(* IEC 61131-3 sources: ironplc-benchmarks/compat_out (part 63) *)

*)

(* @END_DECLARATION := '0' *)
IF A = 0.0 THEN
	TRIANGLE_A := SQRT((s1+s2+S3) * (s1+s2-S3) * (S2+S3-S1) * (S3+S1-S2)) * 0.25;
ELSE
	TRIANGLE_A := S1 * S2 * SIN(RAD(A)) * 0.5;
END_IF;

(* revision histroy
hm	16. oct 2007	rev 1.0
	original version

hm	22. feb 2008	rev 1.1
	improved performance

hm	10. mar. 2009	rev 1.2
	changed syntax of real constants to 0.0

*)
END_FUNCTION

(* @NESTEDCOMMENTS := 'Yes' *)
(* @PATH := '\/Mathematical\/Vektormathematik' *)
(* @OBJECTFLAGS := '0, 8' *)
(* @SYMFILEFLAGS := '2048' *)
FUNCTION V3_ABS : REAL
VAR_INPUT
	A : Vector_3;
END_VAR

(*
version 1.0	11 dec 2007
programmer 	hugo
tested by		tobias

this function calculates the length of a vectors in a 3 dimensional space

*)
(* @END_DECLARATION := '0' *)
V3_ABS := SQRT(A.X * A.X + A.Y * A.Y + A.Z * A.Z);

(* revision history
hm		11 dec 2007	rev 1.0
	original version

*)
END_FUNCTION

(* @NESTEDCOMMENTS := 'Yes' *)
(* @PATH := '\/Mathematical\/Vektormathematik' *)
(* @OBJECTFLAGS := '0, 8' *)
(* @SYMFILEFLAGS := '2048' *)
FUNCTION V3_ADD : vector_3
VAR_INPUT
	A : Vector_3;
	B : Vector_3;
END_VAR

(*
version 1.0	11 dec 2007
programmer 	hugo
tested by		tobias

this function adds two vectors in a 3 dimensional space

*)
(* @END_DECLARATION := '0' *)
V3_ADD.X := A.X + B.X;
V3_ADD.Y := A.Y + B.Y;
V3_ADD.Z := A.Z + B.Z;

(* revision history
hm		11 dec 2007	rev 1.0
	original version

*)
END_FUNCTION

(* @NESTEDCOMMENTS := 'Yes' *)
(* @PATH := '\/Mathematical\/Vektormathematik' *)
(* @OBJECTFLAGS := '0, 8' *)
(* @SYMFILEFLAGS := '2048' *)
FUNCTION V3_ANG : REAL
VAR_INPUT
	A : Vector_3;
	B : Vector_3;
END_VAR
VAR
	d : REAL;
END_VAR

(*
version 1.1	10. mar. 2009
programmer 	hugo
tested by		tobias

this function calculates the angle between two vectors in a 3 dimensional space

*)
(* @END_DECLARATION := '0' *)
d := V3_ABS(A) * V3_ABS(B);
IF d > 0 THEN
	V3_ANG := ACOS(LIMIT(-1.0, V3_DPRO(A, B) / d,1.0));
END_IF;

(* revision history
hm	11. dec. 2007	rev 1.0
	original version

hm	10. mar. 2009	rev 1.1
	changed syntax of real constants to 0.0

*)
END_FUNCTION

(* @NESTEDCOMMENTS := 'Yes' *)
(* @PATH := '\/Mathematical\/Vektormathematik' *)
(* @OBJECTFLAGS := '0, 8' *)
(* @SYMFILEFLAGS := '2048' *)
FUNCTION V3_DPRO : REAL
VAR_INPUT
	A : Vector_3;
	B : Vector_3;
END_VAR

(*
version 1.0	11 dec 2007
programmer 	hugo
tested by		tobias

this function calculates the dot product of two vectors in 3 dimensional space

*)
(* @END_DECLARATION := '0' *)
V3_DPRO := A.X * B.X + A.Y * B.Y + A.Z * B.Z;

(* revision history
hm		11 dec 2007	rev 1.0
	original version

*)
END_FUNCTION

(* @NESTEDCOMMENTS := 'Yes' *)
(* @PATH := '\/Mathematical\/Vektormathematik' *)
(* @OBJECTFLAGS := '0, 8' *)
(* @SYMFILEFLAGS := '2048' *)
FUNCTION V3_NORM : vector_3
VAR_INPUT
	A : Vector_3;
END_VAR
VAR
	la: REAL;
END_VAR

(*
version 1.1	10. mar. 2009
programmer 	hugo
tested by		tobias

this function generates a vectors with absolute length 1 from a vector A in a 3 dimensional space

*)
(* @END_DECLARATION := '0' *)
la := V3_ABS(A);
IF la > 0.0 THEN
	V3_NORM := V3_SMUL(A, 1.0 / la);
END_IF;

(* revision history
hm	11 dec 2007	rev 1.0
	original version

hm	10. mar. 2009	rev 1.1
	changed syntax of real constants to 0.0

*)
END_FUNCTION

(* @NESTEDCOMMENTS := 'Yes' *)
(* @PATH := '\/Mathematical\/Vektormathematik' *)
(* @OBJECTFLAGS := '0, 8' *)
(* @SYMFILEFLAGS := '2048' *)
FUNCTION V3_NUL : BOOL
VAR_INPUT
	A : Vector_3;
END_VAR

(*
version 1.1	10. mar. 2009
programmer 	hugo
tested by		tobias

this function checks if a vectors in a null Vector

*)
(* @END_DECLARATION := '0' *)
V3_NUL := A.X = 0.0 AND A.Y = 0.0 AND A.Z = 0.0;

(* revision history
hm	12 dec 2007	rev 1.0
	original version

hm	10. mar. 2009	rev 1.1
	changed syntax of real constants to 0.0

*)
END_FUNCTION

(* @NESTEDCOMMENTS := 'Yes' *)
(* @PATH := '\/Mathematical\/Vektormathematik' *)
(* @OBJECTFLAGS := '0, 8' *)
(* @SYMFILEFLAGS := '2048' *)
FUNCTION V3_PAR : BOOL
VAR_INPUT
	A : Vector_3;
	B : Vector_3;
END_VAR

(*
version 1.1	10. mar. 2009
programmer 	hugo
tested by		tobias

this function checks if two vectors in a 3 dimensional space are parallel.
which means the two vectors have the same direction

*)
(* @END_DECLARATION := '0' *)
V3_PAR := V3_ABS(V3_XPRO(A, B)) = 0.0;

(* revision history
hm	11 dec 2007	rev 1.0
	original version

hm	10. mar. 2009	rev 1.1
	changed syntax of real constants to 0.0

*)
END_FUNCTION

(* @NESTEDCOMMENTS := 'Yes' *)
(* @PATH := '\/Mathematical\/Vektormathematik' *)
(* @OBJECTFLAGS := '0, 8' *)
(* @SYMFILEFLAGS := '2048' *)
FUNCTION V3_REV : vector_3
VAR_INPUT
	A : Vector_3;
END_VAR

(*
version 1.0	11 dec 2007
programmer 	hugo
tested by		tobias

this function reverses a vector in a 3 dimensional space

*)
(* @END_DECLARATION := '0' *)
V3_REV.X := -A.X;
V3_REV.Y := -A.Y;
V3_REV.Z := -A.Z;

(* revision history
hm		11 dec 2007	rev 1.0
	original version

*)
END_FUNCTION

(* @NESTEDCOMMENTS := 'Yes' *)
(* @PATH := '\/Mathematical\/Vektormathematik' *)
(* @OBJECTFLAGS := '0, 8' *)
(* @SYMFILEFLAGS := '2048' *)
FUNCTION V3_SMUL : vector_3
VAR_INPUT
	A : Vector_3;
	M : REAL;
END_VAR

(*
version 1.0	11 dec 2007
programmer 	hugo
tested by		tobias

this function multiplies a vectors in a 3 dimensional space with a skalar M

*)
(* @END_DECLARATION := '0' *)
V3_SMUL.X := A.X * M;
V3_SMUL.Y := A.Y * M;
V3_SMUL.Z := A.Z * M;

(* revision history
hm		11 dec 2007	rev 1.0
	original version

*)
END_FUNCTION

(* @NESTEDCOMMENTS := 'Yes' *)
(* @PATH := '\/Mathematical\/Vektormathematik' *)
(* @OBJECTFLAGS := '0, 8' *)
(* @SYMFILEFLAGS := '2048' *)
FUNCTION V3_SUB : vector_3
VAR_INPUT
	A : Vector_3;
	B : Vector_3;
END_VAR

(*
version 1.0	11 dec 2007
programmer 	hugo
tested by		tobias

this function subtracts two vectors in a 3 dimensional space
V3_SUB = A - B

*)
(* @END_DECLARATION := '0' *)
V3_SUB.X := A.X - B.X;
V3_SUB.Y := A.Y - B.Y;
V3_SUB.Z := A.Z - B.Z;

(* revision history
hm		11 dec 2007	rev 1.0
	original version

*)
END_FUNCTION

(* @NESTEDCOMMENTS := 'Yes' *)
(* @PATH := '\/Mathematical\/Vektormathematik' *)
(* @OBJECTFLAGS := '0, 8' *)
(* @SYMFILEFLAGS := '2048' *)
FUNCTION V3_XANG : REAL
VAR_INPUT
	A : Vector_3;
END_VAR
VAR
	la: REAL;
END_VAR

(*
version 1.1	10. mar. 2009
programmer 	hugo
tested by		tobias

this function calculates the angle between the X-axis and a vectors in a 3 dimensional space

*)
(* @END_DECLARATION := '0' *)
la := V3_ABS(a);
IF la > 0.0 THEN
	V3_XANG := ACOS(A.X / la);
END_IF;

(* revision history
hm	11 dec 2007	rev 1.0
	original version

hm	10. mar. 2009	rev 1.1
	changed syntax of real constants to 0.0

*)
END_FUNCTION

(* @NESTEDCOMMENTS := 'Yes' *)
(* @PATH := '\/Mathematical\/Vektormathematik' *)
(* @OBJECTFLAGS := '0, 8' *)
(* @SYMFILEFLAGS := '2048' *)
FUNCTION V3_XPRO : vector_3
VAR_INPUT
	A : Vector_3;
	B : Vector_3;
END_VAR

(*
version 1.0	11 dec 2007
programmer 	hugo
tested by		tobias

this function adds two vectors in a 3 dimensional space

*)
(* @END_DECLARATION := '0' *)
V3_XPRO.X := A.Y * B.Z - A.Z * B.Y;
V3_XPRO.Y := A.Z * B.X - A.X * B.Z;
V3_XPRO.Z := A.X * B.Y - A.Y * B.X;

(* revision history
hm		11 dec 2007	rev 1.0
	original version

*)
END_FUNCTION

(* @NESTEDCOMMENTS := 'Yes' *)
(* @PATH := '\/Mathematical\/Vektormathematik' *)
(* @OBJECTFLAGS := '0, 8' *)
(* @SYMFILEFLAGS := '2048' *)
FUNCTION V3_YANG : REAL
VAR_INPUT
	A : Vector_3;
END_VAR
VAR
	la: REAL;
END_VAR

(*
version 1.1	10. mar. 2009
programmer 	hugo
tested by		tobias

this function calculates the angle between the Y-axis and a vectors in a 3 dimensional space

*)
(* @END_DECLARATION := '0' *)
la := V3_ABS(a);
IF la > 0.0 THEN
	V3_YANG := ACOS(A.Y / la);
END_IF;

(* revision history
hm	11 dec 2007	rev 1.0
	original version

hm	10. mar. 2009	rev 1.1
	changed syntax of real constants to 0.0

*)
END_FUNCTION

(* @NESTEDCOMMENTS := 'Yes' *)
(* @PATH := '\/Mathematical\/Vektormathematik' *)
(* @OBJECTFLAGS := '0, 8' *)
(* @SYMFILEFLAGS := '2048' *)
FUNCTION V3_ZANG : REAL
VAR_INPUT
	A : Vector_3;
END_VAR
VAR
	la: REAL;
END_VAR

(*
version 1.1	10. mar. 2009
programmer 	hugo
tested by		tobias

this function calculates the angle between the Z-axis and a vectors in a 3 dimensional space

*)
(* @END_DECLARATION := '0' *)
la := V3_ABS(a);
IF la > 0.0 THEN
	V3_ZANG := ACOS(A.Z / la);
END_IF;

(* revision history
hm	11 dec 2007	rev 1.0
	original version

hm	10. mar. 2009	rev 1.1
	changed syntax of real constants to 0.0

*)
END_FUNCTION

(* @NESTEDCOMMENTS := 'Yes' *)
(* @PATH := '\/Mathematical' *)
(* @OBJECTFLAGS := '0, 8' *)
(* @SYMFILEFLAGS := '2048' *)
FUNCTION ACOSH : REAL
VAR_INPUT
	X : REAL;
END_VAR

(*
version 1.3	10. mar. 2009
programmer 	hugo
tested by		tobias

this function calculates the arcus cos hyperbolicus

*)
(* @END_DECLARATION := '0' *)
ACOSH := LN(SQRT(X * X - 1.0) + X);

(* revision history
hm		12 jan 2007	rev 1.0
	original version

hm		2. dec 2007	rev 1.1
	changed code for better performance

hm	16. mar. 2007		rev 1.2
	changed sequence of calculations to improve performance

hm	10. mar. 2009		rev 1.3
	real constants updated to new systax using dot

*)
END_FUNCTION

(* @NESTEDCOMMENTS := 'Yes' *)
(* @PATH := '\/Mathematical' *)
(* @OBJECTFLAGS := '0, 8' *)
(* @SYMFILEFLAGS := '2048' *)
FUNCTION ACOTH : REAL
VAR_INPUT
	X : REAL;
END_VAR

(*
version 1.2	10. mar. 2009
programmer 	hugo
tested by		tobias

this function calculates the arcus cotangens hyperbolicus

*)
(* @END_DECLARATION := '0' *)
ACOTH := LN((x+1.0)/(x-1.0))*0.5;

(* revision history
hm		12 jan 2007	rev 1.0
	original version

hm		5. jan 2008	rev 1.1
	improved code for better performance

hm	10. mar. 2009		rev 1.2
	real constants updated to new systax using dot

*)
END_FUNCTION

(* @NESTEDCOMMENTS := 'Yes' *)
(* @PATH := '\/Mathematical' *)
(* @OBJECTFLAGS := '0, 8' *)
(* @SYMFILEFLAGS := '2048' *)
FUNCTION AGDF : REAL
VAR_INPUT
	X : REAL;
END_VAR

(*
version 1.1	10. mar. 2009
programmer 	hugo
tested by		tobias

this function calculates the inverse Gudermannian function.

*)
(* @END_DECLARATION := '0' *)
AGDF := LN((1.0 + SIN(X)) / COS(X));

(* comment
the current implementation gives sufficient accuracy only up to X = 1.57 or an output > 10.
is X closer to PI/2 then the function is more and more unreliable
*)

(* revision history
hm	27. apr. 2008	rev 1.0
	original version

hm	10. mar. 2009	rev 1.1
	real constants updated to new systax using dot

*)

END_FUNCTION

(* @NESTEDCOMMENTS := 'Yes' *)
(* @PATH := '\/Mathematical' *)
(* @OBJECTFLAGS := '0, 8' *)
(* @SYMFILEFLAGS := '2048' *)
FUNCTION ASINH : REAL
VAR_INPUT
	X : REAL;
END_VAR

(*
version 1.3	10. mar 2009
programmer 	hugo
tested by		tobias

this function calculates the arcus sin hyperbolicus

*)
(* @END_DECLARATION := '0' *)
ASINH := LN(SQRT(X * X + 1.0)+X);

(* revision history
hm		12 jan 2007	rev 1.0
	original version

hm		2. dec 2007	rev 1.1
	changed code for better performance

hm		16.3. 2007		rev 1.2
	changed sequence of calculations to improve performance

hm	10. mar. 2009		rev 1.3
	real constants updated to new systax using dot

*)
END_FUNCTION

(* @NESTEDCOMMENTS := 'Yes' *)
(* @PATH := '\/Mathematical' *)
(* @OBJECTFLAGS := '0, 8' *)
(* @SYMFILEFLAGS := '2048' *)
FUNCTION ATANH : REAL
VAR_INPUT
	X : REAL;
END_VAR

(*
version 1.2	10. mar. 2009
programmer 	hugo
tested by		tobias

this function calculates the arcus tangens hyperbolicus

*)
(* @END_DECLARATION := '0' *)
ATANH := LN((1.0 + x)/(1.0 - x)) * 0.5;

(* revision history
hm		12 jan 2007	rev 1.0
	original version

hm		5. jan 2008	rev 1.1
	improved code for better performance

hm	10. mar. 2009		rev 1.2
	real constants updated to new systax using dot

*)

END_FUNCTION

(* @NESTEDCOMMENTS := 'Yes' *)
(* @PATH := '\/Mathematical' *)
(* @OBJECTFLAGS := '0, 8' *)
(* @SYMFILEFLAGS := '2048' *)
FUNCTION BETA : REAL
VAR_INPUT
	X : REAL;
	Y : REAL;
END_VAR

(*
version 1.0	26. oct. 2008
programmer 	hugo
tested by		oscat

this function calculates the beta function for real number > 0.

*)
(* @END_DECLARATION := '0' *)
BETA := GAMMA(X) * GAMMA(Y) / GAMMA(x + y);

(* revision history
hm	26. oct. 2008	rev 1.0
	original version

*)
END_FUNCTION

(* @NESTEDCOMMENTS := 'Yes' *)
(* @PATH := '\/Mathematical' *)
(* @OBJECTFLAGS := '0, 8' *)
(* @SYMFILEFLAGS := '2048' *)
FUNCTION BINOM : DINT
VAR_INPUT
	N : INT;
	K : INT;
END_VAR

VAR
	i: INT;
END_VAR

(*
version 1.0	25. oct. 2008
programmer 	hugo
tested by		tobias

this function calculates the binomialkoefficient (N over k)

*)
(* @END_DECLARATION := '0' *)
IF 2 * K > n THEN
	k := n - k;
END_IF;
IF k > n THEN
	RETURN;
ELSIF k = 0 OR k = n THEN
	BINOM := 1;
ELSIF k = 1 THEN
	BINOM := n;
ELSE
	BINOM := n;
	n := n + 1;
	FOR i := 2 TO k DO
		BINOM := BINOM * (n - i) / i;
	END_FOR;
END_IF;

(*
binomialkoeffizient(n, k)
1  wenn k = 0 return 1
2  wenn 2k > n
3      dann f�hre aus ergebnis \leftarrow binomialkoeffizient(n, n-k)
4  sonst f�hre aus ergebnis \leftarrow n
5          von i \leftarrow 2 bis k
6              f�hre aus ergebnis \leftarrow ergebnis \cdot (n + 1 - i)
7                        ergebnis \leftarrow ergebnis : i
8  return ergebnis
*)

(* revision history
hm	25. oct. 2008	rev 1.0
	original version

*)
END_FUNCTION

(* @NESTEDCOMMENTS := 'Yes' *)
(* @PATH := '\/Mathematical' *)
(* @OBJECTFLAGS := '0, 8' *)
(* @SYMFILEFLAGS := '2048' *)
FUNCTION CAUCHY : REAL
VAR_INPUT
	X : REAL;
	T : REAL;
	U : REAL;
END_VAR
VAR
	tmp: REAL;
END_VAR

(*
version 1.0	26. oct. 2008
programmer 	hugo
tested by		tobias

this function calculates the Cauchy distribution function

*)
(* @END_DECLARATION := '0' *)
tmp := x - t;
CAUCHY := math.PI_INV * U / (U*U + tmp*tmp);

(* revision hisdtory
hm	26. oct. 2008	rev 1.0
	original version

*)
END_FUNCTION

(* @NESTEDCOMMENTS := 'Yes' *)
(* @PATH := '\/Mathematical' *)
(* @OBJECTFLAGS := '0, 8' *)
(* @SYMFILEFLAGS := '2048' *)
FUNCTION CAUCHYCD : REAL
VAR_INPUT
	X : REAL;
	T : REAL;
	U : REAL;
END_VAR

(*
version 1.0	26. oct. 2008
programmer 	hugo
tested by		tobias

this function calculates the Cauchy distribution function

*)
(* @END_DECLARATION := '0' *)
CAUCHYCD := 0.5 + math.PI_INV * ATAN((X - T) / U);

(* revision hisdtory
hm	26. oct. 2008	rev 1.0
	original version

*)
END_FUNCTION

(* @NESTEDCOMMENTS := 'Yes' *)
(* @PATH := '\/Mathematical' *)
(* @OBJECTFLAGS := '0, 8' *)
(* @SYMFILEFLAGS := '2048' *)
FUNCTION CEIL : INT
VAR_INPUT
	X : REAL;
END_VAR

(*
version 1.1	21. mar. 2008
programmer 	hugo
tested by	tobias

This is a rounding function which returns the smallest possible integer which is greater or equal to X.
ceil(3.14) = 4
ceil(-3.14) = -3

*)

(* @END_DECLARATION := '0' *)
CEIL := REAL_TO_INT(x);
IF CEIL < X THEN
	CEIL := CEIL + 1;
END_IF;

(* revision history
hm	7. feb. 2007	rev 1.0
	original version

hm	21. mar. 2008	rev 1.1
	use REAL_TO_INT instead of trunc for compatibility reasons

*)

END_FUNCTION

(* @NESTEDCOMMENTS := 'Yes' *)
(* @PATH := '\/Mathematical' *)
(* @OBJECTFLAGS := '0, 8' *)
(* @SYMFILEFLAGS := '2048' *)
FUNCTION CEIL2 : DINT
VAR_INPUT
	X : REAL;
END_VAR

(*
version 1.3	10. mar. 2009
programmer 	hugo
tested by		tobias

This is a rounding function which returns the smallest possible integer which is greater or equal to X.
ceil2(3.14) = 4
ceil2(-3.14) = -3

*)

(* @END_DECLARATION := '0' *)
CEIL2 := REAL_TO_DINT(X);
IF DINT_TO_REAL(CEIL2) < X THEN
	CEIL2 := CEIL2 + 1;
END_IF;

(* revision history
hm	21. mar. 2008	rev 1.0
	original version

hm	4. apr. 2008	rev 1.1
	added type conversion to avoid warnings under codesys 3.0

hm	30. jun. 2008	rev 1.2
	added type conversion to avoid warnings under codesys 3.0

hm	10. mar. 2009	rev 1.3
	use correct statement real_to_DINT

*)

END_FUNCTION

(* @NESTEDCOMMENTS := 'Yes' *)
(* @PATH := '\/Mathematical' *)
(* @OBJECTFLAGS := '0, 8' *)
(* @SYMFILEFLAGS := '2048' *)
FUNCTION CMP : BOOL
VAR_INPUT
	X,Y : REAL;
	N : INT;
END_VAR
VAR
	tmp : REAL;
END_VAR

(*
	version 1.1	10. mar. 2009
	programmer 	hugo
	tested by		tobias

this function checks two inputs x and y if they are identical with the first N digits
example : cmp(3.141516,3.141517,6 is true.

*)
(* @END_DECLARATION := '0' *)
tmp := ABS(x);
IF tmp > 0.0 THEN
	tmp := EXP10(INT_TO_REAL(FLOOR(LOG(tmp))-N+1));
ELSE
	tmp := EXP10(tmp);
END_IF;
CMP := ABS(X - Y) < tmp;

(* revision history
hm	12. mar. 2008	rev 1.0
	original version

hm	10. mar. 2009	rev 1.1
	added type conversion for compatibility reasons
*)

END_FUNCTION

(* @NESTEDCOMMENTS := 'Yes' *)
(* @PATH := '\/Mathematical' *)
(* @OBJECTFLAGS := '0, 8' *)
(* @SYMFILEFLAGS := '2048' *)
FUNCTION COSH : REAL
VAR_INPUT
	X : REAL;
END_VAR
VAR
	t: REAL;
END_VAR

(*
version 1.3	10. mar. 2009
programmer 	hugo
tested by		tobias

this function calculates the cos hyperbolicus

*)
(* @END_DECLARATION := '0' *)
T := EXP(X);
COSH := (1.0 / T + T) * 0.5;

(* revision histroy
hm	12.1.2007	rev 1.0
	original version

hm	1.12.2007	rev 1.1
	changed code to improve performance

hm	5. jan 2008	rev 1.2
	further performance improvement

hm	10. mar. 2009	rev 1.3
	real constants updated to new systax using dot
*)
END_FUNCTION

(* @NESTEDCOMMENTS := 'Yes' *)
(* @PATH := '\/Mathematical' *)
(* @OBJECTFLAGS := '0, 8' *)
(* @SYMFILEFLAGS := '2048' *)
FUNCTION COTH : REAL
VAR_INPUT
	X : REAL;
END_VAR

(*
version 1.4	10. mar. 2009
programmer 	hugo
tested by		tobias

this function calculates the cotangens hyperbolicus

*)
(* @END_DECLARATION := '0' *)
IF X > 20.0 THEN
	COTH :=1.0;
ELSIF X < -20.0 THEN
	COTH := -1.0;
ELSE
	COTH := 1.0 + 2.0 / (EXP(X * 2.0) - 1.0);
END_IF;

(* revision histroy
hm		12.1.2007	rev 1.0
	original version

hm	1.12.2007		rev 1.1
	changed code to improve performance

hm	8. jan 2008	rev 1.2
	further improvement in performance

hm	10. mar 2008	rev 1.3
	extended range of valid inputs to +/- INV
	changed formula for better accuracy

hm	10. mar. 2009	rev 1.4
	real constants updated to new systax using dot
*)
END_FUNCTION

(* @NESTEDCOMMENTS := 'Yes' *)
(* @PATH := '\/Mathematical' *)
(* @OBJECTFLAGS := '0, 8' *)
(* @SYMFILEFLAGS := '2048' *)
FUNCTION D_TRUNC : DINT
VAR_INPUT
	X : REAL;
END_VAR

(*
version 1.2	10. mar. 2009
programmer 	hugo
tested by		oscat

d_trunc truncates a real to a dint 1.5 will be 1 and -1.5 will be -1
d_trunc is necessary because many systems do not offer a trunc to a dint
also real_to_dint will not deliver the same result on different systems

*)

(* @END_DECLARATION := '0' *)
D_TRUNC := REAL_TO_DINT(X);
IF X > 0.0 THEN
	IF DINT_TO_REAL(D_TRUNC) > X THEN D_TRUNC := D_TRUNC - 1; END_IF;
ELSE
	IF DINT_TO_REAL(D_TRUNC) < X THEN D_TRUNC := D_TRUNC + 1; END_IF;
END_IF;

(* for systems that support a dint truncation this routine can be replaced by trunc() *)

(* revision history
hm	21. mar. 2008	rev 1.0
	original version

hm	31. oct. 2008	rev 1.1
	optimized performance

hm	10. mar. 2009	rev 1.2
	real constants updated to new systax using dot
*)
END_FUNCTION

(* @NESTEDCOMMENTS := 'Yes' *)
(* @PATH := '\/Mathematical' *)
(* @OBJECTFLAGS := '0, 8' *)
(* @SYMFILEFLAGS := '2048' *)
FUNCTION DEC1 : INT
VAR_INPUT
	X : INT;
	N : INT;
END_VAR

(*
version 1.1	27. oct. 2008
programmer 	hugo
tested by	oscat

This is a decrement function which decrements the variable X by 1 and if 0 is reached, it begins with N-1 again.
_dec1(X,3) will generate 2,1,0,2,...

*)
(* @END_DECLARATION := '0' *)
IF X = 0 THEN
	DEC1 := N - 1;
ELSE
	DEC1 := X - 1;
END_IF;

(* this is a very elegant version but 50% slower
X := (X - 1 + N) MOD N;
*)

(* revision history
hm	13. oct. 2008	rev 1.0
	original version

hm	27. oct. 2008	rev 1.1
	added statement to return value for compatibility reasons

*)
END_FUNCTION

(* @NESTEDCOMMENTS := 'Yes' *)
(* @PATH := '\/Mathematical' *)
(* @OBJECTFLAGS := '0, 8' *)
(* @SYMFILEFLAGS := '2048' *)
FUNCTION DEG : REAL
VAR_INPUT
	rad : REAL;
END_VAR

(*
version 1.2	10. mar. 2009
programmer 	hugo
tested by		tobias

this function converts degrees into Radiant
execution time on wago 750 - 841 =  10  us
*)
(* @END_DECLARATION := '0' *)
DEG := MODR(57.29577951308232 * RAD, 360.0);

(* revision history
hm	4. aug 2006	rev 1.0
	original version

hm 16. oct 2007	rev 1.1
	added modr statement which prohibits deg to become bigger than 360

hm	10. mar. 2009	rev 1.2
	real constants updated to new systax using dot
*)
END_FUNCTION

(* @NESTEDCOMMENTS := 'Yes' *)
(* @PATH := '\/Mathematical' *)
(* @OBJECTFLAGS := '0, 8' *)
(* @SYMFILEFLAGS := '2048' *)
FUNCTION DIFFER : BOOL
VAR_INPUT
	in1 : REAL;
	in2 : REAL;
	X : REAL;
END_VAR

(*
version 1.1	16 mar 2008
programmer 	hugo
tested by		tobias

this function checks if in1 differs more then x from in2
the output is true if abs(in1-in2) > X

*)
(* @END_DECLARATION := '0' *)
DIFFER := ABS(in1 - in2) > X;

(* revision history
hm		8. oct 2006		rev 1.0
	original version

hm		16. mar 2008	rev 1.1
	improverd code for performance

*)
END_FUNCTION

(* @NESTEDCOMMENTS := 'Yes' *)
(* @PATH := '\/Mathematical' *)
(* @OBJECTFLAGS := '0, 8' *)
(* @SYMFILEFLAGS := '2048' *)
FUNCTION ERF : REAL
VAR_INPUT
	X : REAL;
END_VAR
VAR
	x2 : REAL;
	ax2 : REAL;
END_VAR

(*
version 1.3	10. mar. 2009
programmer 	hugo
tested by		tobias

this function calculates the erf (error) function.

*)
(* @END_DECLARATION := '0' *)
x2 := X*X;
ax2 := 0.147 * x2 + 1.0;
ERF := SQRT(1.0 - EXP(-X2 * ((0.27323954473516 + aX2)/(ax2)))) * SGN(x);

(* revision history
hm	7. apr. 2008	rev 1.0
	original version

hm	30. jun. 2008	rev 1.1
	added type conversions to avoid warnings under codesys 3.0

hm	25. oct. 2008	rev 1.2
	new code using new algorithm

hm	10. mar. 2009	rev 1.3
	real constants updated to new systax using dot
*)
END_FUNCTION

(* @NESTEDCOMMENTS := 'Yes' *)
(* @PATH := '\/Mathematical' *)
(* @OBJECTFLAGS := '0, 8' *)
(* @SYMFILEFLAGS := '2048' *)
FUNCTION ERFC : REAL
VAR_INPUT
	X : REAL;
END_VAR

(*
version 1.1	10. mar. 2009
programmer 	hugo
tested by		tobias

this function calculates the inverse erf (error) function.

*)
(* @END_DECLARATION := '0' *)
ERFC := 1.0 - ERF(X);

(* revision history
hm	7. apr. 2008	rev 1.0
	original version

hm	10. mar. 2009	rev 1.1
	real constants updated to new systax using dot

*)
END_FUNCTION

(* @NESTEDCOMMENTS := 'Yes' *)
(* @PATH := '\/Mathematical' *)
(* @OBJECTFLAGS := '0, 8' *)
(* @SYMFILEFLAGS := '2048' *)
FUNCTION EVEN : BOOL
VAR_INPUT
	in : DINT;
END_VAR

(*
version 1.1	1 dec 2007
programmer 	hugo
tested by		tobias

this function chacks an input for even  value
the output is true if the input is even.
execution time on wago 750 - 841 =  10  us
*)
(* @END_DECLARATION := '0' *)
EVEN := NOT in.0;

(* revision history
hm	1. oct 2006	rev 1.0
	ORIGINAL VERSION

hm	01.12.2007	rev 1.1
	changed code for improved performance

hm	21. mar. 2008	rev 1.2
	changed type of input IN from INT to DINT
*)
END_FUNCTION

(* @NESTEDCOMMENTS := 'Yes' *)
(* @PATH := '\/Mathematical' *)
(* @OBJECTFLAGS := '0, 8' *)
(* @SYMFILEFLAGS := '2048' *)
FUNCTION EXP10 : REAL
VAR_INPUT
	X : REAL;
END_VAR

(*
version 1.0	 2 dec 2007
programmer 	hugo
tested by		tobias

this function calculates the exponent to the basis 10
exp10(3) = 1000

*)
(* @END_DECLARATION := '0' *)
EXP10 := EXP(X * 2.30258509299405);

(* revision history
hm	2. dec 2007		rev 1.0
	original version

*)
END_FUNCTION

(* @NESTEDCOMMENTS := 'Yes' *)
(* @PATH := '\/Mathematical' *)
(* @OBJECTFLAGS := '0, 8' *)
(* @SYMFILEFLAGS := '2048' *)
FUNCTION EXPN : REAL
VAR_INPUT
	X : REAL;
	N : INT;
END_VAR
VAR
	sign: BOOL;
END_VAR

(*
version 1.2	10. mar. 2009
programmer 	hugo
tested by		oscat

this function calculates X to the power of N (Y = X^N) whilke N is an integer
especially on CPU's without a floating point unit this algorythm is about 30 times faster then the IEC standard EXPT() Function

*)
(* @END_DECLARATION := '0' *)
sign := n.15;
N := ABS(N);
IF N.0 THEN EXPN := X; ELSE EXPN := 1.0; END_IF;
N := SHR(N,1);
WHILE N > 0 DO
   X := X * X;
   IF N.0 THEN EXPN := EXPN * X; END_IF;
   N := SHR(N,1);
END_WHILE;
IF sign THEN EXPN := 1.0 / EXPN; END_IF;

(* revision history
hm	4. dec 2007	rev 1.0
	original version

hm	22. oct. 2008	rev 1.1
	optimized code

hm	10. mar. 2009	rev 1.2
	removed nested comments
	real constants updated to new systax using dot

*)
END_FUNCTION

(* @NESTEDCOMMENTS := 'Yes' *)
(* @PATH := '\/Mathematical' *)
(* @OBJECTFLAGS := '0, 8' *)
(* @SYMFILEFLAGS := '2048' *)
FUNCTION FACT : DINT
VAR_INPUT
	X : INT;
END_VAR

(*
version 1.5	26. mar. 2011
programmer 	hugo
tested by		tobias

this function calculates the factorial of x

if the input is negative or higher then 12 the output will be -1.

*)
(* @END_DECLARATION := '0' *)
IF X >= 0 AND X <= 12 THEN
	FACT := math.FACTS[X];
ELSE
	FACT := -1;
END_IF;

(* working code without array
IF X > 12 OR X < 0 THEN
	FACT := -1;
ELSIF X < 7 THEN
	FACT := 1;
	FOR i := 2 TO X DO
		FACT := FACT * i;
	END_FOR;
ELSE
	FACT := 5040;
	FOR i := 8 TO X DO
		FACT := FACT * i;
	END_FOR;
END_IF;
*)

(* revision history
hm 4.3.2007		rev 1.1
	changed a critical error where while loop was indefinite.

hm	10.12.2007	rev 1.2
	start value for i has changed to 2 for better performance

hm	10. mar 2008	rev 1.3
	changed output of fact to dint to allow bigger values

hm	27. oct. 2008	rev 1.4
	optimized code

hm	26. mar. 2011	rev 1.5
	using array math.facts
*)
END_FUNCTION

(* @NESTEDCOMMENTS := 'Yes' *)
(* @PATH := '\/Mathematical' *)
(* @OBJECTFLAGS := '0, 8' *)
(* @SYMFILEFLAGS := '2048' *)
FUNCTION FIB : DINT
VAR_INPUT
	X : INT;
END_VAR
VAR
	t1, t2: DINT;
END_VAR

(*
version 1.3	26. mar. 2008
programmer 	hugo
tested by		tobias

this function calculates the fibonacci sequence

*)
(* @END_DECLARATION := '0' *)
IF X < 0 OR X > 46 THEN
	FIB := -1;
ELSIF x < 2 THEN
	FIB := X;
	RETURN;
ELSE
	(* the fibonacci number is the sum of the two suceeding fibonaci numbers *)
	(* we store the numbers alternatively in t1 and t2 depending on pt *)
	t2 := 1;
	WHILE X > 3 DO
		X := X-2;
		t1 := t1 + t2;
		t2 := t1 + t2;
	END_WHILE;
	IF X > 2 THEN t1 := t1 + t2; END_IF;
	fib := t1 + t2;
END_IF;

(* alternative code for very big numbers

IF X < 31 THEN
	fib := 0.4472136 * (expn(1.618034,X) - expn(-0.618034,X));
ELSE
	fib := 0.4472133 * expn(1.618034,X);
END_IF;

*)

(* revision history
hm		27. dec 2007	rev 1.0
	original version

hm		2. jan 2008	rev 1.1
	deleted unused variable pt

hm		10. mar 2008	rev 1.2
	changed output to dint instead of real

hm		26. mar. 2008	rev 1.3
	function now returns -1 for input < 0 or > 46

*)
END_FUNCTION

(* @NESTEDCOMMENTS := 'Yes' *)
(* @PATH := '\/Mathematical' *)
(* @OBJECTFLAGS := '0, 8' *)
(* @SYMFILEFLAGS := '2048' *)
FUNCTION FLOOR : INT
VAR_INPUT
	X : REAL;
END_VAR

(*
version 1.1	21. mar. 2008
programmer 	hugo
tested by		tobias

This is a rounding function which returns the biggest possible integer which is less or equal to X.
floor(3.14) = 3
floor(-3.14) = -4

*)

(* @END_DECLARATION := '0' *)
FLOOR := REAL_TO_INT(X);
IF FLOOR > X THEN
	FLOOR := FLOOR - 1;
END_IF;

(* revision history
hm		7. feb 2007		rev 1.0
	originlal version

hm		21. mar. 2008	rev 1.1
	replaced trunc with real_to_int for compatibility reasons

*)
END_FUNCTION

(* @NESTEDCOMMENTS := 'Yes' *)
(* @PATH := '\/Mathematical' *)
(* @OBJECTFLAGS := '0, 8' *)
(* @SYMFILEFLAGS := '2048' *)
FUNCTION FLOOR2 : DINT
VAR_INPUT
	X : REAL;
END_VAR

(*
version 1.1	4. apr. 2008
programmer 	hugo
tested by		tobias

This is a rounding function which returns the biggest possible integer which is less or equal to X.
floor2(3.14) = 3
floor2(-3.14) = -4

*)

(* @END_DECLARATION := '0' *)
FLOOR2 := REAL_TO_DINT(X);
IF DINT_TO_REAL(FLOOR2) > X THEN
	FLOOR2 := FLOOR2 - 1;
END_IF;

(* revision history
hm	21. mar. 2008	rev 1.0
	originlal version

hm	4. apr. 2008	rev 1.1
	added type conversion to avoid warnings under codesys 3.0
*)
END_FUNCTION

(* @NESTEDCOMMENTS := 'Yes' *)
(* @PATH := '\/Mathematical' *)
(* @OBJECTFLAGS := '0, 8' *)
(* @SYMFILEFLAGS := '2048' *)
FUNCTION FRACT : REAL
VAR_INPUT
	x : REAL;
END_VAR

(*
version 1.3	10. mar. 2009
programmer 	hugo
tested by		tobias

this function returns the fraction of a real number
fract(3.14) = 0.14

*)
(* @END_DECLARATION := '0' *)
IF ABS(x) < 2.0E9 THEN
	FRACT := x - DINT_TO_REAL(D_TRUNC(x));
ELSE
	FRACT := 0.0;
END_IF;

(* revision history
hm	4. aug 2006	rev 1.0
	original version

hm	11. mar 2008	rev 1.1
	added dint_to_real for compatibility reasons
	now returns 0 for number > 2e9
	changed input to x

hm	21. mar. 2008	rev 1.2
	use D_trunc instead of TRUNC for compatibility reasons

hm	10. mar. 2009	rev 1.3
	real constants updated to new systax using dot

*)
END_FUNCTION

(* @NESTEDCOMMENTS := 'Yes' *)
(* @PATH := '\/Mathematical' *)
(* @OBJECTFLAGS := '0, 8' *)
(* @SYMFILEFLAGS := '2048' *)
FUNCTION GAMMA : REAL
VAR_INPUT
	X : REAL;
END_VAR

(*
version 1.3	10. mar. 2009
programmer 	hugo
tested by		oscat

this function calculates the stirling function which is an approximation for the gamma function

*)
(* @END_DECLARATION := '0' *)
IF x > 0.0 THEN
	GAMMA := SQRT(math.PI2 / X) * EXPT(math.E_INV * (x + 1.0 / (12.0 * x - 0.1 / X)), X);
END_IF;

(* the stirling formula is not very accurate for small values of X
IF X >=0 THEN GAMMA := SQRT(math.PI2 * X) * EXPT(X / math.E, X); END_IF;
*)

(* revision history
hm	10.12.2007	rev 1.0
	original version

hm	18. oct. 2008	rev 1.1
	using math constants

hm	26. oct. 2008	rev 1.2
	using new formula with better accuracy

hm	10. mar. 2009	rev 1.3
	real constants updated to new systax using dot

*)
END_FUNCTION

(* @NESTEDCOMMENTS := 'Yes' *)
(* @PATH := '\/Mathematical' *)
(* @OBJECTFLAGS := '0, 8' *)
(* @SYMFILEFLAGS := '2048' *)
FUNCTION GAUSS : REAL
VAR_INPUT
	X : REAL;
	U : REAL;
	SI: REAL;
END_VAR
VAR
	temp: REAL;
	si_inv: REAL;
END_VAR

(*
version 1.2	10. mar. 2009
programmer 	hugo
tested by		tobias

this function calculates the gaussian density function

*)
(* @END_DECLARATION := '0' *)
temp := X - U;
si_inv := 1.0  / si;
GAUSS := EXP(Temp * Temp * si_inv * si_inv * - 0.5) * 0.39894228 * si_inv;

(* revision hisdtory
hm	6. apr. 2008	rev 1.0
	original version

hm	27. oct. 2008	rev 1.1
	optimized performance

hm	10. mar. 2009	rev 1.2
	real constants updated to new systax using dot

*)
END_FUNCTION

(* @NESTEDCOMMENTS := 'Yes' *)
(* @PATH := '\/Mathematical' *)
(* @OBJECTFLAGS := '0, 8' *)
(* @SYMFILEFLAGS := '2048' *)
FUNCTION GAUSSCD : REAL
VAR_INPUT
	X : REAL;
	U : REAL;
	SI: REAL;
END_VAR

(*
version 1.1	10. mar. 2009
programmer 	hugo
tested by		tobias

this function calculates the gaussian cumulative distribution function

*)
(* @END_DECLARATION := '0' *)
GAUSSCD := (ERF((X - U) / (SI * 1.414213562)) + 1.0) * 0.5;

(* revision hisdtory
hm	6. apr. 2008	rev 1.0
	original version

hm	10. mar. 2009	rev 1.1
	real constants updated to new systax using dot

*)
END_FUNCTION

(* @NESTEDCOMMENTS := 'Yes' *)
(* @PATH := '\/Mathematical' *)
(* @OBJECTFLAGS := '0, 8' *)
(* @SYMFILEFLAGS := '2048' *)
FUNCTION GCD : INT
VAR_INPUT
	A : DINT;
	B : DINT;
END_VAR
VAR
	t: DINT;
END_VAR

(*
version 1.0	19. jan. 2011
programmer 	hugo
tested by	tobias

this function calculates the gretaest common divisor of two numbers A and B

*)
(* @END_DECLARATION := '0' *)
IF A = 0 THEN
	GCD := DINT_TO_INT(ABS(B));
ELSIF B = 0 THEN
	GCD := DINT_TO_INT(ABS(A));
ELSE
	A := ABS(A);
	B := ABS(B);
	GCD := 1;
	WHILE NOT(A.0 OR B.0) DO
		A := SHR(A,1);
		B := SHR(B,1);
		GCD := SHL(GCD,1);
	END_WHILE;
	WHILE A > 0 DO
		IF NOT(A.0) THEN A := SHR(A,1);
		ELSIF NOT(B.0) THEN B := SHR(B,1);
		ELSE
			t:= SHR(ABS(A-B),1);
			IF A < B THEN B := t; ELSE A := T; END_IF;
		END_IF;
	END_WHILE;
	GCD := GCD * DINT_TO_INT(B);
END_IF;

(* revision history
hm	19. jan. 2011	rev 1.0
	original version

*)
END_FUNCTION

(* @NESTEDCOMMENTS := 'Yes' *)
(* @PATH := '\/Mathematical' *)
(* @OBJECTFLAGS := '0, 8' *)
(* @SYMFILEFLAGS := '2048' *)
FUNCTION GDF : REAL
VAR_INPUT
	X : REAL;
END_VAR

(*
version 1.2	10. mar. 2009
programmer 	hugo
tested by		tobias

this function calculates the Gudermannian function.

*)
(* @END_DECLARATION := '0' *)
IF X = 0.0 THEN
	GDF := 0.0;
ELSIF X > 15.0 THEN
	GDF := math.PI05;
ELSIF X < -15.0 THEN
	GDF := -math.PI05;
ELSE
	GDF := ATAN(EXP(X)) * 2.0 - math.PI05;
END_IF;

(* revision history
hm	27. apr. 2008	rev 1.0
	original version

hm	18. oct. 2008	rev 1.1
	using math constants

hm	10. mar. 2009	rev 1.2
	real constants updated to new systax using dot

*)

END_FUNCTION

(* @NESTEDCOMMENTS := 'Yes' *)
(* @PATH := '\/Mathematical' *)
(* @OBJECTFLAGS := '0, 8' *)
(* @SYMFILEFLAGS := '2048' *)
FUNCTION GOLD : REAL
VAR_INPUT
	X : REAL;
END_VAR

(*
version 1.1	10. mar. 2009
programmer 	hugo
tested by		tobias

this function calculates the golden function.

*)
(* @END_DECLARATION := '0' *)
GOLD := (X + SQRT(X*X + 4.0)) * 0.5;

(* revision history
hm	27. apr. 2008	rev 1.0
	original version

hm	10. mar. 2009	rev 1.1
	real constants updated to new systax using dot

*)

END_FUNCTION

(* @NESTEDCOMMENTS := 'Yes' *)
(* @PATH := '\/Mathematical' *)
(* @OBJECTFLAGS := '0, 8' *)
(* @SYMFILEFLAGS := '2048' *)
FUNCTION HYPOT : REAL
VAR_INPUT
	X : REAL;
	Y : REAL;
END_VAR

(*
version 1.0	21 feb 2008
programmer 	hugo
tested by	oscat

this function calculates the pythagorean function

*)
(* @END_DECLARATION := '0' *)
HYPOT := SQRT(x*x + y*y);

(* revision history
hm	21. feb 2008	rev 1.0
	original version

*)

END_FUNCTION

(* @NESTEDCOMMENTS := 'Yes' *)
(* @PATH := '\/Mathematical' *)
(* @OBJECTFLAGS := '0, 8' *)
(* @SYMFILEFLAGS := '2048' *)
FUNCTION INC : INT
VAR_INPUT
	X : INT;
	D : INT;
	M : INT;
END_VAR

(*
version 1.1	15. jan 2008
programmer 	hugo
tested by	oscat

This is a increment function which increments the input X by the value D and compares the result with M.
if the output exceeds M it will continue to count from 0 again.

*)
(* @END_DECLARATION := '0' *)
INC := (X + D + M + 1) MOD (M + 1);

(* revision history
hm	7. feb 2007		REV 1.0
	original version

hm	15. jan 2008	rev 1.1
	allow for neagtive increment

*)
END_FUNCTION

(* @NESTEDCOMMENTS := 'Yes' *)
(* @PATH := '\/Mathematical' *)
(* @OBJECTFLAGS := '0, 8' *)
(* @SYMFILEFLAGS := '2048' *)
FUNCTION INC1 : INT
VAR_INPUT
	X : INT;
	N : INT;
END_VAR

(*
version 1.2	23. feb. 2009
programmer 	hugo
tested by	oscat

This is a increment function which increments the variable X by 1 and if N is reached, it begins with 0 instead of N again.
inc1(X,3) will generate 0,1,2,0,1,.....

*)
(* @END_DECLARATION := '0' *)
IF X >= N - 1 THEN
	INC1 := 0;
ELSE
	INC1 := X + 1;
END_IF;

(* revision history
hm	13. oct. 2008	rev 1.0
	original version

hm	22. oct. 2008	rev 1.1
	added statement to return value for compatibility reasons

hm	23. feb. 2009	rev 1.2
 	when inc1 is called with X >= N inc will continue with 0
*)
END_FUNCTION

(* @NESTEDCOMMENTS := 'Yes' *)
(* @PATH := '\/Mathematical' *)
(* @OBJECTFLAGS := '0, 8' *)
(* @SYMFILEFLAGS := '2048' *)
FUNCTION INC2 : INT
VAR_INPUT
	X : INT;
	D : INT;
	L : INT;
	U : INT;
END_VAR
VAR
	tmp: INT;
END_VAR

(*
version 1.0	29. jun. 2008
programmer 	hugo
tested by	oscat

This function increments the input X by the value D and compares the result with U.
if the output exceeds U it will continue to count from L again.

*)
(* @END_DECLARATION := '0' *)
tmp := U - L + 1;
INC2 := (X + D - L + tmp) MOD tmp + L;

(* revision history
hm	29. jun. 2008		REV 1.0
	original version

*)
END_FUNCTION

(* @NESTEDCOMMENTS := 'Yes' *)
(* @PATH := '\/Mathematical' *)
(* @OBJECTFLAGS := '0, 8' *)
(* @SYMFILEFLAGS := '2048' *)
FUNCTION INV : REAL
VAR_INPUT
	X : REAL;
END_VAR

(*
version 1.1	10. mar. 2009
programmer 	hugo
tested by		tobias

This function calculates the result of 1 / X

*)

(* @END_DECLARATION := '0' *)
IF X <> 0.0 THEN INV := 1.0 / X; END_IF;

(* revision history
hm	26. oct. 2008	rev 1.0
	original version

hm	10. mar. 2009	rev 1.1
	real constants updated to new systax using dot

*)

END_FUNCTION

(* @NESTEDCOMMENTS := 'Yes' *)
(* @PATH := '\/Mathematical' *)
(* @OBJECTFLAGS := '0, 8' *)
(* @SYMFILEFLAGS := '2048' *)
FUNCTION LAMBERT_W : REAL
VAR_INPUT
	X : REAL;
END_VAR
VAR
	w : REAL;
	i : INT;
	we: REAL;
	w1e: REAL;
	last: DWORD;
	ewx: REAL;
END_VAR

(*
version 1.1	10. mar. 2009
programmer 	hugo
tested by		oscat

this function calculates the lambert_w function.

*)
(* @END_DECLARATION := '0' *)
(* check for valid input and return -1000 if too low *)
IF x < -0.367879441171442 THEN
	LAMBERT_W := -1000.0;
	RETURN;
(* return 0 if x = 0 *)
ELSIF x = 0.0 THEN
	RETURN;
(* first an estimate is calculated *)
ELSIF x <= 500.0 THEN
	w := LN(x + 1.0);
	w := 0.665 * (1.0 + 0.0195 * w) * w + 0.04;
ELSE
	w := LN(x - 4.0) - (1.0 - 1.0/LN(x)) * LN(LN(x));
END_IF;
(* use estimate to calculate exact result *)
FOR i := 0 TO 5 DO
	ewx := EXP(w);
	we := w * ewx - x;
	w1e := (w+1.0) * ewx;
	last := REAL_TO_DW(w) AND 16#FFFF_FFFC;
	w := w - (we / (w1e - (w+2.0) * we / (2.0 * w + 2.0)));
	IF (REAL_TO_DW(w) AND 16#FFFF_FFFC) = last THEN EXIT; END_IF;
END_FOR;
LAMBERT_W := w;

(* revision hisdtory
hm	26. oct. 2008	rev 1.0
	original version

hm	10. mar. 2009	rev 1.1
	real constants updated to new systax using dot

*)
END_FUNCTION

(* @NESTEDCOMMENTS := 'Yes' *)
(* @PATH := '\/Mathematical' *)
(* @OBJECTFLAGS := '0, 8' *)
(* @SYMFILEFLAGS := '2048' *)
FUNCTION LANGEVIN : REAL
VAR_INPUT
	X : REAL;
END_VAR

(*
version 1.2	10.mar. 2009
programmer 	hugo
tested by		tobias

this function calculates the langevin function

*)
(* @END_DECLARATION := '0' *)
IF X = 0.0 THEN
	LANGEVIN := 0.0;
ELSE
	LANGEVIN := COTH(X) - 1.0 / X;
END_IF;

(* revision history
hm	10.12.2007	rev 1.0
	original version

hm	11. mar 2008	rev 1.1
	changed formula to avoid problems when x = 0

hm	10. mar. 2009	rev 1.2
	real constants updated to new systax using dot

*)
END_FUNCTION

(* @NESTEDCOMMENTS := 'Yes' *)
(* @PATH := '\/Mathematical' *)
(* @OBJECTFLAGS := '0, 8' *)
(* @SYMFILEFLAGS := '2048' *)
FUNCTION MAX3 : REAL
VAR_INPUT
	in1 : REAL;
	in2 : REAL;
	in3 : REAL;
END_VAR

(*
version 1.1	18. mar. 2011
programmer 	hugo
tested by		tobias

this function returns the highest of 3 real values

*)
(* @END_DECLARATION := '0' *)
MAX3 := MAX(MAX(IN1,IN2),IN3);

(* revision history
hm	1.1.2007	rev 1.0
	original release

hm	18. mar. 2011	rev 1.1
	improve performance

*)
END_FUNCTION

(* @NESTEDCOMMENTS := 'Yes' *)
(* @PATH := '\/Mathematical' *)
(* @OBJECTFLAGS := '0, 8' *)
(* @SYMFILEFLAGS := '2048' *)
FUNCTION MID3 : REAL
VAR_INPUT
	IN1 : REAL;
	IN2 : REAL;
	IN3 : REAL;
END_VAR

(*
version 1.2	18. mar. 2011
programmer 	hugo
tested by		tobias

returns the mid value of 3 real inputs.

*)

(* @END_DECLARATION := '0' *)
IF IN1 > IN2 THEN MID3 := IN1; IN1 := IN2; IN2 := MID3; END_IF;
IF IN2 > IN3 THEN IN2 := IN3; END_IF;
MID3 := SEL(IN1 > IN2, IN2, IN1);

(*
hm	1.1.2007	rev 1.1
	rewrote the function for better performance

hm	18. mar. 2011	rev 1.2
	improve performance
*)
END_FUNCTION

(* @NESTEDCOMMENTS := 'Yes' *)
(* @PATH := '\/Mathematical' *)
(* @OBJECTFLAGS := '0, 8' *)
(* @SYMFILEFLAGS := '2048' *)
FUNCTION MIN3 : REAL
VAR_INPUT
	in1 : REAL;
	in2 : REAL;
	in3 : REAL;
END_VAR

(*
version 1.1	18. mar. 2011
programmer 	hugo
tested by		tobias

this function returns the lowest of 3 real values

*)
(* @END_DECLARATION := '0' *)
MIN3 := MIN(MIN(IN1,IN2),IN3);

(* revision history
hm	1.1.2007	rev 1.0
	original release

hm	18. mar. 2011	rev 1.1
	improve performance

*)
END_FUNCTION

(* @NESTEDCOMMENTS := 'Yes' *)
(* @PATH := '\/Mathematical' *)
(* @OBJECTFLAGS := '0, 8' *)
(* @SYMFILEFLAGS := '2048' *)
FUNCTION MODR : REAL
VAR_INPUT
	IN : REAL;
	DIVI : REAL;
END_VAR

(*
version 1.5	10. mar. 2009
programmer 	hugo
tested by		tobias

this is a modulo funtion for real numbers
modr(5.5,2.5) = 0.5

*)

(* @END_DECLARATION := '0' *)
IF divi = 0.0 THEN
	MODR := 0.0;
ELSE
	MODR := in - DINT_TO_REAL(FLOOR2(in / divi)) * divi;
END_IF;

(* revision history

hm	4. aug.2006		rev 1.0

hm	28. jan.2007	rev 1.1
	modr(x,0) will deliver the result 0

hm	21. mar 2008	rev 1.2
	use D_trunc for compatibility reasons

hm	4. apr. 2008	rev 1.3
	added type conversion to avoid warnings under codesys 3.0

hm	31. oct. 2008	rev 1.4
	changed algorithm to the more common version using floor instead of TRUNC

hm	10. mar. 2009	rev 1.5
	real constants updated to new systax using dot

*)
END_FUNCTION

(* @NESTEDCOMMENTS := 'Yes' *)
(* @PATH := '\/Mathematical' *)
(* @OBJECTFLAGS := '0, 8' *)
(* @SYMFILEFLAGS := '2048' *)
FUNCTION MUL_ADD : REAL
VAR_INPUT
	X : REAL;
	K : REAL;
	O : REAL;
END_VAR

(*
version 1.1	11 nov 2007
programmer 	hugo
tested by		tobias

this function multiplies an input X with K and adds Offset O to the result.

*)
(* @END_DECLARATION := '0' *)
MUL_ADD := X * K + O;

(* revision history
hm	28. feb 2007
	original version

hm	11.nov 2007		rev 1.1
	deleted preset values for K and O this makes no sense for a function

*)
END_FUNCTION

(* @NESTEDCOMMENTS := 'Yes' *)
(* @PATH := '\/Mathematical' *)
(* @OBJECTFLAGS := '0, 8' *)
(* @SYMFILEFLAGS := '2048' *)
FUNCTION NEGX : REAL
VAR_INPUT
	X : REAL;
END_VAR

(*
version 1.0	26. oct. 2008
programmer 	hugo
tested by	tobias

This function returns -X

*)

(* @END_DECLARATION := '0' *)
NEGX := -X;

(* revision history
hm	26. oct. 2008	rev 1.0
	original version

*)

END_FUNCTION

(* @NESTEDCOMMENTS := 'Yes' *)
(* @PATH := '\/Mathematical' *)
(* @OBJECTFLAGS := '0, 8' *)
(* @SYMFILEFLAGS := '2048' *)
FUNCTION RAD : REAL
VAR_INPUT
	DEG : REAL;
END_VAR

(*
version 1.2	18. oct. 2008
programmer 	hugo
tested by	tobias

this function converts Radiant to degrees

*)
(* @END_DECLARATION := '0' *)
RAD := MODR(0.0174532925199433 * DEG, math.PI2);

(* revision history
hm	4. aug 2006		rev 1.0
	original version

hm 	16. oct 2007	rev 1.1
	added modr statement which prohibits rad to become bigger than 2PI

hm	18. oct 2008	rev 1.2
	using math constants

*)
END_FUNCTION

(* @NESTEDCOMMENTS := 'Yes' *)
(* @PATH := '\/Mathematical' *)
(* @OBJECTFLAGS := '0, 8' *)
(* @SYMFILEFLAGS := '2048' *)
FUNCTION RDM : REAL
VAR_INPUT
	last : REAL;
END_VAR
VAR
	tn : DWORD;
	tc : INT;
END_VAR

(*
version 1.9	10. mar. 2009
programmer 	hugo
tested by		tobias

this function calculates a pseudo random number
to generate the number it reads the sps timer and calculates a random number between 0 and 1:
in order to use rdm more then once within one sps cycle it need to be called with different seed numbers LAST.

*)
(* @END_DECLARATION := '0' *)
tn := T_PLC_MS();
tc := BIT_COUNT(tn);
tn.31 := tn.2;
tn.30 := tn.5;
tn.29 := tn.4;
tn.28 := tn.1;
tn.27 := tn.0;
tn.26 := tn.7;
tn.25 := tn.6;
tn.24 := tn.3;
tn := ROL(tn,BIT_COUNT(tn)) OR 16#80000001;
tn := tn MOD 71474513 + INT_TO_DWORD(tc + 77);
RDM := FRACT(DWORD_TO_REAL(tn) / 10000000.0 * (math.E - LIMIT(0.0,last,1.0)));

(*
pt := REF(temp);
pt^ := (T_PLC_MS() AND 16#007FFFFF) OR 16#3D000000;
RDM := fract(modR(temp*e+pi1, PI1-last) + modR(temp*PI1+e + last,e-last));
*)

(* revision history
hm		16. jan 2007		rev 1.0
	original version

hm		11. nov 2007		rev 1.1
	changed time() into t_plc_ms()

hm		20. nov 2007		rev 1.2
	changed code of temp calculation to avoid overflow in modr due to resuclt would not fit DINT for high timeer values

hm		5. jan 2008		rev 1.3
	changed calculation of temp to avoid problem with high values of t_plc_ms

hm		2. feb 2008		rev 1.4
	changed algorithm to avoind non iec functions and guarantee more randomness

hm	10. mar. 2008		rev 1.5
	make sure last will be between 0 and 1 to avoid invalid results

hm	16. mar. 2008		rev 1.6
	added conversion for tc to avoid warnings under codesys 3.0

hm	18. may. 2008		rev 1.7
	changed constant E to E1

hm	18. oct. 2008		rev 1.8
	using math constants

hm	10. mar. 2009		rev 1.9
	real constants updated to new systax using dot

*)
END_FUNCTION

(* @NESTEDCOMMENTS := 'Yes' *)
(* @PATH := '\/Mathematical' *)
(* @OBJECTFLAGS := '0, 8' *)
(* @SYMFILEFLAGS := '2048' *)
FUNCTION RDM2 : INT
VAR_INPUT
	last : INT;
	low : INT;
	high : INT;
END_VAR

(*
version 1.1	18. oct. 2008
programmer 	hugo
tested by	tobias

this function calculates an integer pseudo random number
the random number will be in the range of low <= rdm2 <= high.

*)
(* @END_DECLARATION := '0' *)
RDM2 := TRUNC(RDM(FRACT(last * math.PI)) * (high - low + 1)) + low;

(* revision history
hm		29. feb 2008		rev 1.0
	original version

hm		18. oct. 2008		rev 1.1
	using math constants

*)
END_FUNCTION

(* @NESTEDCOMMENTS := 'Yes' *)
(* @PATH := '\/Mathematical' *)
(* @OBJECTFLAGS := '0, 8' *)
(* @SYMFILEFLAGS := '2048' *)
FUNCTION RDMDW : DWORD
VAR_INPUT
	last : DWORD;
END_VAR
VAR
	RX: REAL;
	M: REAL;
END_VAR

(*
version 1.2	18. oct. 2008
programmer 	hugo
tested by		tobias

this function calculates a DWORD pseudo random number.

*)
(* @END_DECLARATION := '0' *)
M := BIT_COUNT(last);
RX := RDM(FRACT(M * math.PI));
RDMDW := SHL(REAL_TO_DWORD(rx*65535),16);
RX := RDM(FRACT(M * math.E));
RDMDW := RDMDW OR (REAL_TO_DWORD(rx*65535) AND 16#0000FFFF);

(* revision history
hm		14. mar 2008		rev 1.0
	original version

hm		18. may. 2008		rev 1.1
	changed constant E to E1

hm		18. oct. 2008		rev 1.2
	using math constants

*)
END_FUNCTION

(* @NESTEDCOMMENTS := 'Yes' *)
(* @PATH := '\/Mathematical' *)
(* @OBJECTFLAGS := '0, 8' *)
(* @SYMFILEFLAGS := '2048' *)
FUNCTION REAL_TO_FRAC : FRACTION
VAR_INPUT
	X : REAL;					(* in einen Bruch umzuwandelnder Wert *)
	N : INT;					(* maximale Gr��e des Nenners *)
END_VAR
VAR
	temp : DINT;				(* Merker f�r Berechnungen *)

	sign: BOOL;					(* Vorzeichen vom Eingangswert *)
	X_gerundet: DINT;			(* Wert von Bruch, auf ganze Zahl gerundet *)
	X_ohne_Nachkomma: REAL;		(* Wert von Bruch, ohne Nachkommastellen *)
	Numerator:       DINT := 1;	(* Initialwert Zaehler  *)
	Denominator:     DINT := 0;	(* Initialwert Nenner *)
	Numerator_old:   DINT := 0;	(* Initialwert Zaehler der letzten Berechnung  *)
	Denominator_old: DINT := 1;	(* Initialwert Zaehler der letzten Berechnung   *)

END_VAR

(*
version 1.1		06. apr. 2011
programmer 	alexander
tested by		hugo

this function calculates the closest fraction for a real number

*)

(* @END_DECLARATION := '0' *)
IF X < 0.0 THEN
	sign := TRUE;								(* Vorzeichen merken *)
	X := ABS(X);								(* Absolutwert berechnen *)
END_IF;

REPEAT
	X_gerundet := REAL_TO_DINT(X);

	(* Zaehler berechnen *)
	temp := numerator * X_gerundet + numerator_old;		(* Zaehler um Vorkammawert erweitern *)
	numerator_old := numerator;							(* Zaehler der letzten Berechnung speichern *)
	numerator := temp;									(* Zaehler dieser Berechnung speichern *)

	(* Nenner berechnen *)
	temp := denominator * X_gerundet + denominator_old;	(* Nenner um Vorkammawert erweitern *)
	denominator_old := denominator;						(* Nenner der letzten Berechnung speichern *)
	denominator := temp;								(* Nenner dieser Berechnung speichern *)

	(* Restwert berechnen *)
	X_ohne_Nachkomma := DINT_TO_REAL(X_gerundet);
	IF X = X_ohne_Nachkomma THEN						(* Bruch geht ohne Rest auf *)
		IF ABS(denominator) <= N THEN						(* kein Rundungsfehler *)
			numerator_old := numerator;					(* Numerator_old wird von Funktion zur�ckgegeben *)
			denominator_old := denominator;			(* Denominator_old wird von Funktion zur�ckgegeben *)
		END_IF
		EXIT;											(* keine weitere Berechnung notwendig *)
	ELSE
		X := 1.0 / (X - X_ohne_Nachkomma);				(* Kehrwert vom Rest -> Neuer Bruch *)
	END_IF

UNTIL
	ABS(Denominator) > N
END_REPEAT

(* correct sign if X was negative *)
IF sign THEN
	REAL_TO_FRAC.NUMERATOR := -1 * ABS(DINT_TO_INT(numerator_old));
ELSE
	REAL_TO_FRAC.NUMERATOR :=  ABS(DINT_TO_INT(numerator_old));
END_IF
REAL_TO_FRAC.DENOMINATOR := ABS(DINT_TO_INT(denominator_old));

(* revision history
hm		19. jan. 2011	rev 1.0
	original version

ad		06. apr. 2011	rev 1.1
	optimized code
*)
END_FUNCTION

(* @NESTEDCOMMENTS := 'Yes' *)
(* @PATH := '\/Mathematical' *)
(* @OBJECTFLAGS := '0, 8' *)
(* @SYMFILEFLAGS := '2048' *)
FUNCTION RND : REAL
VAR_INPUT
	X : REAL;
	N : INT;
END_VAR
VAR
	M : REAL;
END_VAR

(*
version 1.2	10. mar. 2009
programmer 	hugo
tested by		tobias

this function rounds a real down to n digits total.
round(3.1415,2) = 3.1

*)
(* @END_DECLARATION := '0' *)
IF X = 0.0 THEN
	RND := 0.0;
ELSE
	M := EXPN(10.0,N - CEIL(LOG(ABS(X))));
	RND := DINT_TO_REAL(REAL_TO_DINT(X * M)) / M;
END_IF;

(* revision history
hm	11. mar 2008	rev 1.0
	original version

hm	26. oct. 2008	rev 1.1
	code optimization

hm	10. mar. 2009	rev 1.2
	real constants updated to new systax using dot

*)

END_FUNCTION

(* @NESTEDCOMMENTS := 'Yes' *)
(* @PATH := '\/Mathematical' *)
(* @OBJECTFLAGS := '0, 8' *)
(* @SYMFILEFLAGS := '2048' *)
FUNCTION SGN : INT
VAR_INPUT
	X : REAL;
END_VAR

(*
version 1.1	11. nov. 2008
programmer 	hugo
tested by	tobias

sgn returns 0 when X = 0 , -1 when X < 1 and +1 when X > 1

*)

(* @END_DECLARATION := '0' *)
IF X > 0 THEN
	SGN := 1;
ELSIF X < 0 THEN
	SGN := -1;
ELSE
	SGN := 0;
END_IF;

(* revision histroy
hm	16. oct 2007	rev 1.0
	original version

hm	11. nov 2007	rev 1.1
	changed type of function from real to int

*)
END_FUNCTION

(* @NESTEDCOMMENTS := 'Yes' *)
(* @PATH := '\/Mathematical' *)
(* @OBJECTFLAGS := '0, 8' *)
(* @SYMFILEFLAGS := '2048' *)
FUNCTION SIGMOID : REAL
VAR_INPUT
	X : REAL;
END_VAR

(*
version 1.2	10. mar. 2009
programmer 	hugo
tested by		tobias

this function calculates the sigmoid function

*)
(* @END_DECLARATION := '0' *)
IF X > 20.0 THEN
	SIGMOID := 1.0;
ELSIF x < -85.0 THEN
	SIGMOID := 0.0;
ELSE
	SIGMOID := 1.0 / (1.0 + EXP(-X));
END_IF;

(* revision history
hm	10.12.2007		rev 1.0
	original version

hm	11. mar. 2008		rev 1.1
	extended range of valid inputs to +inv / -inv

hm 10. mar. 2009		rev 1.2
	real constants updated to new systax using dot

*)
END_FUNCTION

(* @NESTEDCOMMENTS := 'Yes' *)
(* @PATH := '\/Mathematical' *)
(* @OBJECTFLAGS := '0, 8' *)
(* @SYMFILEFLAGS := '2048' *)
FUNCTION SIGN_I : BOOL
VAR_INPUT
	IN : DINT;
END_VAR

(*
version 1.3	27. oct. 2008
programmer 	hugo
tested by	tobias

this function return true if the integer input is negative

*)
(* @END_DECLARATION := '0' *)
SIGN_I := in.31;

(* revision history
hm 3.3.2007	rev 1.1
	changed method of function for better compatibility to other systems

hm	1.12.2007	rev 1.2
	changed code to improve performance

hm	27. oct. 2008	rev 1.3
	changed type of input to dint

*)
END_FUNCTION

(* @NESTEDCOMMENTS := 'Yes' *)
(* @PATH := '\/Mathematical' *)
(* @OBJECTFLAGS := '0, 8' *)
(* @SYMFILEFLAGS := '2048' *)
FUNCTION SIGN_R : BOOL
VAR_INPUT
	in : REAL;
END_VAR

(*
version 1.4	10. mar. 2009
programmer 	hugo
tested by		tobias

this function return true if the real input is negative

*)
(* @END_DECLARATION := '0' *)
SIGN_R := in < 0.0;

(* revision history
hm 19.1.2007	rev 1.1
	changed method of function for better compatibility to other systems

hm	1.12.2007	rev 1.2
	changed code to improve performance

hm	14. jun. 2008	rev 1.3
	improved performace

hm 10. mar. 2009	rev 1.4
	real constants updated to new systax using dot

*)
END_FUNCTION

(* @NESTEDCOMMENTS := 'Yes' *)
(* @PATH := '\/Mathematical' *)
(* @OBJECTFLAGS := '0, 8' *)
(* @SYMFILEFLAGS := '2048' *)
FUNCTION SINC : REAL
VAR_INPUT
	X : REAL;
END_VAR

(*
version 1.2	10. mar. 2009
programmer 	hugo
tested by		tobias

this function calculates the sinc function.

*)
(* @END_DECLARATION := '0' *)
IF X = 0.0 THEN
	SINC := 1.0;
ELSE
	SINC := SIN(x) / x;
END_IF;

(* revision histroy
hm	11. mar. 2008	rev 1.0
	original version

hm	1.12.2007	rev 1.1
	changed code to improove performance

hm 10. mar. 2009	rev 1.2
	real constants updated to new systax using dot

*)
END_FUNCTION

(* @NESTEDCOMMENTS := 'Yes' *)
(* @PATH := '\/Mathematical' *)
(* @OBJECTFLAGS := '0, 8' *)
(* @SYMFILEFLAGS := '2048' *)
FUNCTION SINH : REAL
VAR_INPUT
	X : REAL;
END_VAR

(*
version 1.3	11. mar 2008
programmer 	hugo
tested by		tobias

this function calculates the sin hyperbolicus

*)
(* @END_DECLARATION := '0' *)
IF ABS(x) < 2E-3 THEN
	SINH := X;
ELSE
	SINH := (EXP(x) - EXP(-x)) * 0.5;
END_IF;

(* revision history
hm	12.1.2007	rev 1.0
	original version

hm	1.12.2007	rev 1.1
	changed code to improve performance

hm	5. jan 2008	rev 1.2
	further performance improvement

hm	11. mar 2008	rev 1.3
	improved accuracy around 0

*)
END_FUNCTION

(* @NESTEDCOMMENTS := 'Yes' *)
(* @PATH := '\/Mathematical' *)
(* @OBJECTFLAGS := '0, 8' *)
(* @SYMFILEFLAGS := '2048' *)
FUNCTION SQRTN : REAL
VAR_INPUT
	X : REAL;
	N : INT;
END_VAR

(*
version 1.3	10. mar. 2009
programmer 	hugo
tested by		tobias

this function calculates the nth root function of X according to the formula sqrtn = x^(1/n).

*)
(* @END_DECLARATION := '0' *)
IF N > 0 THEN
	SQRTN := EXP(LN(x) / INT_TO_REAL(n));
ELSE
	SQRTN := 0.0;
END_IF;

(* revision history
hm		12 jan 2007	rev 1.0
	original version

hm		2. dec 2007	rev 1.1
	changed code for better performance

hm		11. mar 2008	rev 1.2
	added result 0 for compatibility reasons

hm 10. mar. 2009	rev 1.3
	added type conversions for compatibility reasons

*)
END_FUNCTION

(* @NESTEDCOMMENTS := 'Yes' *)
(* @PATH := '\/Mathematical' *)
(* @OBJECTFLAGS := '0, 8' *)
(* @SYMFILEFLAGS := '2048' *)
FUNCTION TANC : REAL
VAR_INPUT
	X : REAL;
END_VAR

(*
version 1.1	10. mar. 2009
programmer 	hugo
tested by		oscat

this function calculates the tanc function.

*)
(* @END_DECLARATION := '0' *)
IF X = 0.0 THEN
	TANC := 1.0;
ELSE
	TANC := TAN(x) / x;
END_IF;

(* revision histroy
hm	23. oct. 2008	rev 1.0
	original version

hm 10. mar. 2009	rev 1.1
	real constants updated to new systax using dot

*)
END_FUNCTION

(* @NESTEDCOMMENTS := 'Yes' *)
(* @PATH := '\/Mathematical' *)
(* @OBJECTFLAGS := '0, 8' *)
(* @SYMFILEFLAGS := '2048' *)
FUNCTION TANH : REAL
VAR_INPUT
	X : REAL;
END_VAR

(*
version 1.3	10. mar. 2009
programmer 	hugo
tested by		tobias

this function calculates the tangens hyperbolicus

*)
(* @END_DECLARATION := '0' *)
IF X > 20.0 THEN
	TANH := 1.0;
ELSIF X < -20.0 THEN
	TANH := -1.0;
ELSE
	TANH := 1.0 - 2.0 / (EXP(2.0 * x) + 1.0);
END_IF;

(* revision hisdtory
hm		12.1.2007		rev 1.0
	original version

hm		1.12.2007		rev 1.1
	changed code to improve performance

hm		10. mar 2008	rev 1.2
	corrected an error in formula
	extended range of valid inputs to +/- INV

hm 10. mar. 2009	rev 1.3
	real constants updated to new systax using dot

*)
END_FUNCTION

(* @NESTEDCOMMENTS := 'Yes' *)
(* @PATH := '\/Mathematical' *)
(* @OBJECTFLAGS := '0, 8' *)
(* @SYMFILEFLAGS := '2048' *)
FUNCTION WINDOW : BOOL
VAR_INPUT
	low : REAL;
	in : REAL;
	high : REAL;
END_VAR

(*
	version 1.1	22 jan 2007
	programmer 	hugo
	tested BY	tobias

this checks a signal if the signal is between the upper and lower limit
*)
(* @END_DECLARATION := '0' *)
WINDOW := in < high AND in > low;

(* revision history
hm	22.1.2007	rev 1.1
	changed the order of inputs to low, in, high

*)
END_FUNCTION

(* @NESTEDCOMMENTS := 'Yes' *)
(* @PATH := '\/Mathematical' *)
(* @OBJECTFLAGS := '0, 8' *)
(* @SYMFILEFLAGS := '2048' *)
FUNCTION WINDOW2 : BOOL
VAR_INPUT
	LOW : REAL;
	IN : REAL;
	HIGH : REAL;
END_VAR

(*
	version 1.0	31 oct 2007
	programmer 	hugo
	tested BY	tobias

this checks a signal if the signal is between the upper and lower limit including the two limits
*)
(* @END_DECLARATION := '0' *)
WINDOW2 := IN >= LOW AND IN <= HIGH;

(* revision history
hm	31.10.2007	rev 1.0
	original version

*)
END_FUNCTION

(* @NESTEDCOMMENTS := 'Yes' *)
(* @PATH := '\/Other' *)
(* @OBJECTFLAGS := '0, 8' *)
(* @SYMFILEFLAGS := '2048' *)
FUNCTION_BLOCK ESR_COLLECT
VAR_INPUT
	ESR_0, ESR_1, ESR_2, ESR_3, ESR_4, ESR_5, ESR_6, ESR_7 : ARRAY [0..3] OF esr_data;
	rst : BOOL;
END_VAR
VAR_IN_OUT
	pos : INT;
END_VAR
VAR_OUTPUT
	ESR_OUT : ARRAY[0..31] OF esr_data;
END_VAR
VAR CONSTANT
	max_in : INT := 3; (* max limit of input array *)
	max_out : INT := 32; (* number of elements in array *)
END_VAR
VAR
	cnt : INT := -1;
END_VAR

(*
version 1.4	1. dec. 2009
programmer 	hugo
tested by		tobias

ESR_collect collects esr data from up to 8 esr_mon modules and stroes them in an output array.
the output pos will display the position of the last element in the array. if the array is empty, pos = -1
when to buffer is read by followon modules. pos has to be reset to -1
if the array will be full, the buffer will be refilled starting at position 0.

*)

(* @END_DECLARATION := '0' *)
IF rst OR cnt < 0 THEN
	pos := -1;
ELSE
	FOR cnt := 0 TO max_in DO
	IF esr_0[cnt].typ > 0 THEN pos := INC1(pos, max_out); esr_out[pos] := esr_0[cnt]; END_IF;
	IF esr_1[cnt].typ > 0 THEN pos := INC1(pos, max_out); esr_out[pos] := esr_1[cnt]; END_IF;
	IF esr_2[cnt].typ > 0 THEN pos := INC1(pos, max_out); esr_out[pos] := esr_2[cnt]; END_IF;
	IF esr_3[cnt].typ > 0 THEN pos := INC1(pos, max_out); esr_out[pos] := esr_3[cnt]; END_IF;
	IF esr_4[cnt].typ > 0 THEN pos := INC1(pos, max_out); esr_out[pos] := esr_4[cnt]; END_IF;
	IF esr_5[cnt].typ > 0 THEN pos := INC1(pos, max_out); esr_out[pos] := esr_5[cnt]; END_IF;
	IF esr_6[cnt].typ > 0 THEN pos := INC1(pos, max_out); esr_out[pos] := esr_6[cnt]; END_IF;
	IF esr_7[cnt].typ > 0 THEN pos := INC1(pos, max_out); esr_out[pos] := esr_7[cnt]; END_IF;
   END_FOR;
END_IF;

(* revision history
hm	26.jan 2007	rev 1.0
	original version

hm	8. dec 2007	rev 1.1
	added reset input

ks	27. oct. 2008	rev 1.2
	optimized code for performance

ks	12. nov. 2009	rev 1.3
	output pos was not pointing to last value

hm	1. dec. 2009	rev 1.4
	changed pos to be I/O
	reduced output array size to 32 elements
*)
END_FUNCTION_BLOCK

(* @NESTEDCOMMENTS := 'Yes' *)
(* @PATH := '\/Other' *)
(* @OBJECTFLAGS := '0, 8' *)
(* @SYMFILEFLAGS := '2048' *)
FUNCTION_BLOCK ESR_MON_B8
VAR_INPUT
	s0, s1, s2, s3, s4, s5, s6, s7 : BOOL;
	DT_in : DT;
END_VAR
VAR_INPUT (* CONSTANT *)
	a0, a1, a2, a3, a4, a5, a6, a7 : STRING[10];
END_VAR
VAR_OUTPUT
	ESR_Flag : BOOL;
END_VAR
VAR_IN_OUT
	ESR_Out: ARRAY [0..3] OF esr_data;
END_VAR
VAR
	x0, x1, x2, x3, x4, x5, x6, x7 : BOOL;
	tx: TIME;
	cnt : INT;
END_VAR

(*
version 1.3	1. dec. 2009
programmer 	hugo
tested by		tobias

ESR_mon_B8 monitores up to 8 binary inputs and reports changes with time stamd and adress label.
the module checks 8 inputs for a change and reports all changes with time and adress stamp to the output.
4 events maximum can be collected at once within the same cycle

*)

(* @END_DECLARATION := '0' *)
(* read system timer *)
tx := DWORD_TO_TIME(T_PLC_MS());

ESR_Flag := FALSE;
esr_out[3].typ := 0;
esr_out[2].typ := 0;
esr_out[1].typ := 0;
esr_out[0].typ := 0;
cnt := 0;

(* check if inputs have chaged and fill buffer *)
IF s0 <> X0 THEN
	esr_out[cnt].typ := 10 + BOOL_TO_BYTE(s0);
	esr_out[cnt].adress := a0;
	esr_out[cnt].DS := DT_in;
	esr_out[cnt].TS := TX;
	X0 := S0;
	cnt := cnt + 1;
	esr_flag := TRUE;
END_IF;
IF s1 <> X1 THEN
	esr_out[cnt].typ := 10 + BOOL_TO_BYTE(s1);
	esr_out[cnt].adress := a1;
	esr_out[cnt].DS := DT_in;
	esr_out[cnt].TS := TX;
	X1 := S1;
	cnt := cnt + 1;
	esr_flag := TRUE;
END_IF;
IF s2 <> X2 THEN
	esr_out[cnt].typ := 10 + BOOL_TO_BYTE(s2);
	esr_out[cnt].adress := a2;
	esr_out[cnt].DS := DT_in;
	esr_out[cnt].TS := TX;
	X2 := S2;
	cnt := cnt + 1;
	esr_flag := TRUE;
END_IF;
IF s3 <> X3 THEN
	esr_out[cnt].typ := 10 + BOOL_TO_BYTE(s3);
	esr_out[cnt].adress := a3;
	esr_out[cnt].DS := DT_in;
	esr_out[cnt].TS := TX;
	X3 := S3;
	cnt := cnt + 1;
	esr_flag := TRUE;
END_IF;
IF s4 <> X4 AND cnt < 4 THEN
	esr_out[cnt].typ := 10 + BOOL_TO_BYTE(s4);
	esr_out[cnt].adress := a4;
	esr_out[cnt].DS := DT_in;
	esr_out[cnt].TS := TX;
	X4 := S4;
	cnt := cnt + 1;
	esr_flag := TRUE;
END_IF;
IF s5 <> X5  AND cnt < 4 THEN
	esr_out[cnt].typ := 10 + BOOL_TO_BYTE(s5);
	esr_out[cnt].adress := a5;
	esr_out[cnt].DS := DT_in;
	esr_out[cnt].TS := TX;
	X5 := S5;
	cnt := cnt + 1;
	esr_flag := TRUE;
END_IF;
IF s6 <> X6  AND cnt < 4 THEN
	esr_out[cnt].typ := 10 + BOOL_TO_BYTE(s6);
	esr_out[cnt].adress := a6;
	esr_out[cnt].DS := DT_in;
	esr_out[cnt].TS := TX;
	X6 := S6;
	cnt := cnt + 1;
	esr_flag := TRUE;
END_IF;
IF s7 <> X7  AND cnt < 4 THEN
	esr_out[cnt].typ := 10 + BOOL_TO_BYTE(s7);
	esr_out[cnt].adress := a7;
	esr_out[cnt].DS := DT_in;
	esr_out[cnt].TS := TX;
	X7 := S7;
	cnt := cnt + 1;
	esr_flag := TRUE;
END_IF;

(* revision history
hm	26. jan 2007	rev 1.0
	original version

hm	17. sep 2007	rev 1.1
	replaced time() with T_PLC_MS() for compatibility reasons

hm	22. oct. 2008	rev 1.2
	optimized code

hm	1.dec. 2009	rev 1.3
	changed esr_out to be I/O

*)
END_FUNCTION_BLOCK

(* @NESTEDCOMMENTS := 'Yes' *)
(* @PATH := '\/Other' *)
(* @OBJECTFLAGS := '0, 8' *)
(* @SYMFILEFLAGS := '2048' *)
FUNCTION_BLOCK ESR_MON_R4
VAR_INPUT
	R0, R1, R2, R3 : REAL;
	DT_in : DT;
END_VAR
VAR_INPUT (* CONSTANT *)
	a0, a1, a2, a3 : STRING[10];
	s0, s1, s2, s3 : REAL;
END_VAR
VAR_OUTPUT
	ESR_Flag : BOOL;
END_VAR
VAR_IN_OUT
	ESR_Out: ARRAY [0..3] OF esr_data;
END_VAR
VAR
	p0, p1, p2, p3 : REF_TO DWORD;
	x0, x1, x2, x3 : REAL;
	tx: TIME;
	cnt : INT;
END_VAR

(*
version 1.4	1. dec. 2009
programmer 	hugo
tested by		tobias

ESR_mon_R4 monitores up to 4 Real inputs and reports changes with time stamd and adress label.
the module checks 4 inputs for a change of more than the specified sensitivity S and reports all changes with time and adress stamp to the output.

*)

(* @END_DECLARATION := '0' *)
(* read system timer *)
tx := DWORD_TO_TIME(T_PLC_MS());
P0 := REF(R0);
P1 := REF(R1);
P2 := REF(R2);
P3 := REF(R3);

ESR_Flag := FALSE;
esr_out[3].typ := 0;
esr_out[2].typ := 0;
esr_out[1].typ := 0;
esr_out[0].typ := 0;
cnt := 0;

(* check if inputs have chaged and fill buffer *)
IF DIFFER(R0,  X0, S0) THEN
	esr_out[cnt].typ := 20;
	esr_out[cnt].adress := a0;
	esr_out[cnt].DS := DT_in;
	esr_out[cnt].TS := TX;
	esr_out[cnt].data[0] := Byte_of_Dword(P0^,0);
	esr_out[cnt].data[1] := Byte_of_Dword(P0^,1);
	esr_out[cnt].data[2] := Byte_of_Dword(P0^,2);
	esr_out[cnt].data[3] := Byte_of_Dword(P0^,3);
	X0 := R0;
	cnt := cnt + 1;
	esr_flag := TRUE;
END_IF;
IF differ(R1,  X1, S1) THEN
	esr_out[cnt].typ := 20;
	esr_out[cnt].adress := a1;
	esr_out[cnt].DS := DT_in;
	esr_out[cnt].TS := TX;
	esr_out[cnt].data[0] := Byte_of_Dword(P1^,0);
	esr_out[cnt].data[1] := Byte_of_Dword(P1^,1);
	esr_out[cnt].data[2] := Byte_of_Dword(P1^,2);
	esr_out[cnt].data[3] := Byte_of_Dword(P1^,3);
	X1 := R1;
	cnt := cnt + 1;
	esr_flag := TRUE;
END_IF;
IF differ(R2,  X2, S2) THEN
	esr_out[cnt].typ := 20;
	esr_out[cnt].adress := a2;
	esr_out[cnt].DS := DT_in;
	esr_out[cnt].TS := TX;
	esr_out[cnt].data[0] := Byte_of_Dword(P2^,0);
	esr_out[cnt].data[1] := Byte_of_Dword(P2^,1);
	esr_out[cnt].data[2] := Byte_of_Dword(P2^,2);
	esr_out[cnt].data[3] := Byte_of_Dword(P2^,3);
	X2 := R2;
	cnt := cnt + 1;
	esr_flag := TRUE;
END_IF;
IF DIFFER(R3,  X3, S3) THEN
	esr_out[cnt].typ := 20;
	esr_out[cnt].adress := a3;
	esr_out[cnt].DS := DT_in;
	esr_out[cnt].TS := TX;
	esr_out[cnt].data[0] := Byte_of_Dword(P3^,0);
	esr_out[cnt].data[1] := Byte_of_Dword(P3^,1);
	esr_out[cnt].data[2] := Byte_of_Dword(P3^,2);
	esr_out[cnt].data[3] := Byte_of_Dword(P3^,3);
	X3 := R3;
	cnt := cnt + 1;
	esr_flag := TRUE;
END_IF;

(* revision history
hm	26. jan 2007	rev 1.0
	original version

hm	17. sep. 2007		rev 1.1
	replaced time() with T_PLC_MS() for compatibility reasons

hm	8. dec. 2007		rev 1.2
	corrected an error while esr typ would not be set

hm	16. mar. 2008		rev 1.3
	deleted wrong conversion real_to_dword

hm	1. dec 2009		rev 1.4
	changed esr_out to be I/O

*)

END_FUNCTION_BLOCK

(* @NESTEDCOMMENTS := 'Yes' *)
(* @PATH := '\/Other' *)
(* @OBJECTFLAGS := '0, 8' *)
(* @SYMFILEFLAGS := '2048' *)
FUNCTION_BLOCK ESR_MON_X8
VAR_INPUT
	s0, s1, s2, s3, s4, s5, s6, s7 : BYTE;
	DT_in : DT;
	Mode : BYTE := 3;
END_VAR
VAR_INPUT (* CONSTANT *)
	a0, a1, a2, a3, a4, a5, a6, a7 : STRING[10];
END_VAR
VAR_OUTPUT
	ESR_Flag : BOOL;
END_VAR
VAR_IN_OUT
	ESR_Out: ARRAY [0..3] OF esr_data;
END_VAR
VAR
	x0, x1, x2, x3, x4, x5, x6, x7 : BYTE;
	tx: TIME;
	cnt : INT;
END_VAR

(*
version 1.2	1. dec. 2009
programmer 	hugo
tested by		tobias

ESR_MON_X8 is a status and error collector.
the module checks 8 status inputs for a change and reports up to 4 input changes with time and adress stamp to the output.
the mode can be
1 for error only
2 for error and status
3 for error, status and debug
the adress label of the 8 inputs can be configured individually.
*)

(* @END_DECLARATION := '0' *)
(* read system timer *)
tx := DWORD_TO_TIME(T_PLC_MS());

ESR_Flag := FALSE;
esr_out[3].typ := 0;
esr_out[2].typ := 0;
esr_out[1].typ := 0;
esr_out[0].typ := 0;
cnt := 0;

(* check if inputs have chaged and fill buffer *)
IF s0 <> X0 AND ((s0 < 100) OR (S0 > 99 AND S0 < 200 AND mode >= 2) OR (S0 > 199 AND mode = 3)) THEN
	esr_out[cnt] := status_to_ESR(s0, a0, DT_in, TX);
	X0 := S0;
	cnt := cnt + 1;
	esr_flag := TRUE;
END_IF;
IF s1 <> X1 AND ((s1 < 100) OR (S1 > 99 AND S1 < 200 AND mode >= 2) OR (S1 > 199 AND mode = 3)) THEN
	esr_out[cnt] := status_to_ESR(s1, a1, DT_in, TX);
	X1 := S1;
	cnt := cnt + 1;
	esr_flag := TRUE;
END_IF;
IF s2 <> X2 AND ((s2 < 100) OR (S2 > 99 AND S2 < 200 AND mode >= 2) OR (S2 > 199 AND mode = 3)) THEN
	esr_out[cnt] := status_to_ESR(s2, a2, DT_in, TX);
	X2 := S2;
	cnt := cnt + 1;
	esr_flag := TRUE;
END_IF;
IF s3 <> X3 AND ((s3 < 100) OR (S3 > 99 AND S3 < 200 AND mode >= 2) OR (S3 > 199 AND mode = 3)) THEN
	esr_out[cnt] := status_to_ESR(s3, a3, DT_in, TX);
	X3 := S3;
	cnt := cnt + 1;
	esr_flag := TRUE;
END_IF;
IF cnt < 4 AND s4 <> X4 AND ((s4 < 100) OR (S4 > 99 AND S4 < 200 AND mode >= 2) OR (S4 > 199 AND mode = 3)) THEN
	esr_out[cnt] := status_to_ESR(s4, a4, DT_in, TX);
	X4 := S4;
	cnt := cnt + 1;
	esr_flag := TRUE;
END_IF;
IF cnt < 4 AND s5 <> X5 AND ((s5 < 100) OR (S5 > 99 AND S5 < 200 AND mode >= 2) OR (S5 > 199 AND mode = 3)) THEN
	esr_out[cnt] := status_to_ESR(s5, a5, DT_in, TX);
	X5 := S5;
	cnt := cnt + 1;
	esr_flag := TRUE;
END_IF;
IF cnt < 4 AND s6 <> X6 AND ((s6 < 100) OR (S6 > 99 AND S6 < 200 AND mode >= 2) OR (S6 > 199 AND mode = 3)) THEN
	esr_out[cnt] := status_to_ESR(s6, a6, DT_in, TX);
	X6 := S6;
	cnt := cnt + 1;
	esr_flag := TRUE;
END_IF;
IF cnt < 4 AND s7 <> X7 AND ((s7 < 100) OR (S7 > 99 AND S7 < 200 AND mode >= 2) OR (S7 > 199 AND mode = 3)) THEN
	esr_out[cnt] := status_to_ESR(s7, a7, DT_in, TX);
	X7 := S7;
	cnt := cnt + 1;
	esr_flag := TRUE;
END_IF;

(* revision history
hm	26. jan 2007		rev 1.0
	original version

hm	17. sep 2007	rev 1.1
	replaced time() with T_PLC_MS() for compatibility reasons

hm	1. dec. 2009	rev 1.2
	changed esr_out to be I/O

*)
END_FUNCTION_BLOCK

(* @NESTEDCOMMENTS := 'Yes' *)
(* @PATH := '\/Other' *)
(* @OBJECTFLAGS := '0, 8' *)
(* @SYMFILEFLAGS := '2048' *)
FUNCTION OSCAT_VERSION : DWORD
VAR_INPUT
	IN : BOOL;
END_VAR

(*
version 1.1	16 dec 2007
programmer 	hugo
tested by		oscat

oscat_version returns the version number in dword format
132 is library version 1.32
if IN = true, the release date will be returned

*)
(* @END_DECLARATION := '0' *)
IF in THEN
	OSCAT_VERSION := DATE_TO_DWORD(D#2012-01-02);
ELSE
	OSCAT_VERSION := 333;
END_IF;

(* revision history
hm	6. oct 2006	rev 1.0
	original version

hm	16. dec 2007	rev 1.1
	added possibility to return date and version depending on IN.

*)
END_FUNCTION

(* @NESTEDCOMMENTS := 'Yes' *)
(* @PATH := '\/Other' *)
(* @OBJECTFLAGS := '0, 8' *)
(* @SYMFILEFLAGS := '2048' *)
FUNCTION STATUS_TO_ESR : esr_data
VAR_INPUT
	status : BYTE;
	adress : STRING[10];
	DT_in : DT;
	TS : TIME;
END_VAR

(*
version 1.0	6 oct 2006
programmer 	hugo
tested by		tobias

status_to_esr creates esr data from a status byte.

*)
(* @END_DECLARATION := '0' *)
IF status < 100 THEN
	status_to_ESR.typ := 1;
ELSIF status < 200 THEN
	status_to_ESR.typ := 2;
ELSE
	status_to_ESR.typ := 3;
END_IF;
status_to_ESR.adress:= adress;
status_to_ESR.DS := DT_in;
status_to_ESR.TS := TS;
status_to_ESR.data[0] := status;

END_FUNCTION

(* @NESTEDCOMMENTS := 'Yes' *)
(* @PATH := '\/String' *)
(* @OBJECTFLAGS := '0, 8' *)
(* @SYMFILEFLAGS := '2048' *)
FUNCTION BIN_TO_BYTE : BYTE
VAR_INPUT
	BIN : STRING[12];
END_VAR
VAR
	pt : REF_TO BYTE;
	i: INT;
	X: BYTE;
	stop: INT;
END_VAR

(*
version 1.2	26. jul 2009
programmer 	hugo
tested by		oscat

BINARY_TO_byte converts a binary string into a byte.

*)
(* @END_DECLARATION := '0' *)
pt := REF(bin);
stop := LEN(bin);
FOR I := 1 TO stop DO
	x := pt^;
	(* calculate the value of the digit *)
	IF X = 48 THEN
		BIN_TO_BYTE := SHL(BIN_TO_BYTE,1);
	ELSIF X = 49 THEN
		BIN_TO_BYTE := SHL(BIN_TO_BYTE,1) OR 1;
	END_IF;
	pt := pt + 1;
END_FOR;

(* revision histroy
hm	18. jun. 2008	rev 1.0
	original release

hm	20. sep. 2008	rev 1.1
	changed length of input string from 20 to 12

hm	26. jul. 2009	rev 1.2
	optimized code
*)

END_FUNCTION

(* @NESTEDCOMMENTS := 'Yes' *)
(* @PATH := '\/String' *)
(* @OBJECTFLAGS := '0, 8' *)
(* @SYMFILEFLAGS := '2048' *)
FUNCTION BIN_TO_DWORD : DWORD
VAR_INPUT
	BIN : STRING[40];
END_VAR
VAR
	pt : REF_TO BYTE;
	i: INT;
	X: BYTE;
	stop: INT;
END_VAR

(*
version 1.2	26. jul. 2009
programmer 	hugo
tested by		oscat

BINARY_TO_DWORD converts a binary string into a dword.

*)
(* @END_DECLARATION := '0' *)
pt := REF(bin);
stop := LEN(bin);
FOR I := 1 TO stop DO
	x := pt^;
	(* calculate the value of the digit *)
	IF X = 48 THEN
		BIN_TO_DWORD := SHL(BIN_TO_DWORD,1);
	ELSIF X = 49 THEN
		BIN_TO_DWORD := SHL(BIN_TO_DWORD,1) OR 1;
	END_IF;
	pt := pt + 1;
END_FOR;

(* revision histroy
hm	18. jun. 2008	rev 1.0
	original release

hm	20. sep. 2008	rev 1.1
	changed length of input dtring from 20 to 40

hm	26. jul 2009	rev 1.2
	optimized code
*)

END_FUNCTION

(* @NESTEDCOMMENTS := 'Yes' *)
(* @PATH := '\/String' *)
(* @OBJECTFLAGS := '0, 8' *)
(* @SYMFILEFLAGS := '2048' *)
FUNCTION BYTE_TO_STRB : STRING[8]
VAR_INPUT
	IN : BYTE;
END_VAR
VAR
	i: INT;
	pt : REF_TO BYTE;
END_VAR

(*
version 1.3	20. jun. 2008
programmer 	hugo
tested by	oscat

BYTE_TO_STRINGB converts a Byte to a String of Bits represented by '0' and '1' s.
The lowest order bit will be on the right and the high order bit on the left.

*)

(* @END_DECLARATION := '0' *)
(* pointer f�r die ausgabe ermitteln *)
pt := REF(BYTE_TO_STRB);
(* die 8 ausgabecharacter ermitteln und schreiben *)
FOR i := 1 TO 8 DO
	pt^ := BOOL_TO_BYTE(in.7) + 48;
	in := SHL(in,1);
	pt := pt + 1;
END_FOR;

(* der ausgabestring muss noch mit 0 abgeschlossen werden *)
pt^ := 0;

(* code before rev 1.1
FOR i := 1 TO 8 DO
	IF in.0 = 0 THEN temp := CONCAT('0', temp); ELSE temp := CONCAT('1', temp); END_IF;
	in := SHR(in, 1);
END_FOR;
BYTE_TO_STRB := temp;
*)

(* revision history

hm		9.6.2007	rev 1.0
	original version

hm	15. dec 2007	rev 1.1
	inprooved code for higher performance

hm	29. mar. 2008	rev 1.2
	changed STRING to STRING[8]

hm	20. jun. 2008	rev 1.3
	performance improvement

*)
END_FUNCTION

(* @NESTEDCOMMENTS := 'Yes' *)
(* @PATH := '\/String' *)
(* @OBJECTFLAGS := '0, 8' *)
(* @SYMFILEFLAGS := '2048' *)
FUNCTION BYTE_TO_STRH : STRING[2]
VAR_INPUT
	IN : BYTE;
END_VAR
VAR
	temp : BYTE;
	PT : REF_TO BYTE;
END_VAR

(*
version 1.3	29 mar. 2008
programmer 	hugo
tested by		tobias

BYTE_TO_STRINGH converts a Byte to a String of Hexadecimal represented by '0' .. '9' and 'A' .. 'F'.
The lowest order Character will be on the right and the high order Character on the left.

*)

(* @END_DECLARATION := '0' *)
(* read pointer to output string *)
PT := REF(BYTE_TO_STRH);
(* calculate high order hex value *)
temp := SHR(in,4);
(* convert value to hex character *)
IF temp <= 9 THEN temp := temp + 48; ELSE temp := temp + 55; END_IF;
(* write friat character to output string *)
PT^ := temp;
(* calculate low order hex value *)
temp := in AND 2#00001111;
IF temp <= 9 THEN temp := temp + 48; ELSE temp := temp + 55; END_IF;
(* increment pointer and wirte low order character *)
pt := pt + 1;
pt^ := temp;
(* set pointer at the end of the output string and close the string with 0 *)
pt := pt + 1;
pt^:= 0;

(* code before rev 1.2
FOR i := 1 TO 2 DO
	X := in AND 2#1111;
	IF X <= 9 THEN X := X + 48; ELSE X := X + 55; END_IF;
	Cx := CHR(X);
	temp := CONCAT(Cx, temp);
	in := SHR(in,4);
END_FOR;
BYTE_TO_STRH := temp;
*)

(* revision history

hm	9.6.2007		rev 1.0
	original version

hm	11.9.2007		rev 1.1
	changed coding for compatibility with twincat, under twincat concat cannot have a function as argument.

hm	15 dec 2007		REV 1.2
	changed code for higher performance

hm	29. mar. 2008	rev 1.3
	changed STRING to STRING[2]
*)
END_FUNCTION

(* @NESTEDCOMMENTS := 'Yes' *)
(* @PATH := '\/String' *)
(* @OBJECTFLAGS := '0, 8' *)
(* @SYMFILEFLAGS := '2048' *)
FUNCTION CAPITALIZE : STRING[STRING_LENGTH]
VAR_INPUT
	str : STRING[STRING_LENGTH];
END_VAR
VAR
	PT : REF_TO BYTE;
	pos : INT;
	L : INT;
	first : BOOL := TRUE;
END_VAR

(*
version 1.2	20. jun. 2008
programmer 	hugo
tested by		tobias

capitalize returns str with all first letters after a blank or beginning of the string are converted to uppercase.

*)
(* @END_DECLARATION := '0' *)
PT := REF(CAPITALIZE);
CAPITALIZE := str;
L := LEN(str);
FOR pos := 1 TO l DO
	IF first THEN pt^ := TO_UPPER(pt^);	END_IF;
	(* remember in first if the next char needs to capitalized *)
	first := pt^= 32;
	PT := pt + 1;
END_FOR;

(* revision histroy
hm		4. mar 2008	rev 1.0
	original release

hm	29. mar. 2008	rev 1.1
	changed STRING to STRING[STRING_LENGTH]

hm	20. jun. 2008	rev 1.2
	improved performance

*)

END_FUNCTION

(* @NESTEDCOMMENTS := 'Yes' *)
(* @PATH := '\/String' *)
(* @OBJECTFLAGS := '0, 8' *)
(* @SYMFILEFLAGS := '2048' *)
FUNCTION CHARCODE : BYTE
VAR_INPUT
	STR : STRING[10];
END_VAR
VAR
	found: STRING[1];
	search : STRING[10];
	pos: INT;
	i: INT;
END_VAR

(*
version 1.2		24. oct. 2008
programmer 		hugo
tested by		hugo

CHARCODE converts a HTML Character NAME INTO ITS code
'�uml' is convterted to �
'euro' is converted to �

*)
(* @END_DECLARATION := '0' *)
IF LEN(str) = 1 THEN
	CHARCODE := CODE(STR, 1);
ELSIF str <> '' THEN
	(* construct search string *)
	search := CONCAT('&', str);
	search := CONCAT(search, ';');
	WHILE pos = 0 AND (i < 4) DO
		i := i + 1;
		pos := FIND(setup.CHARNAMES[i], search);
	END_WHILE;
	found := MID(setup.CHARNAMES[i], 1, pos - 1);
	CHARCODE := CODE(found, 1);
END_IF;

(* revision history
hm	13. may. 2008	rev 1.0
	original version

hm	19. oct. 2008	rev 1.1
	changed setup constants

hm	24. oct. 2008	rev 1.2
	optimized code
*)

END_FUNCTION

(* @NESTEDCOMMENTS := 'Yes' *)
(* @PATH := '\/String' *)
(* @OBJECTFLAGS := '0, 8' *)
(* @SYMFILEFLAGS := '2048' *)
FUNCTION CHARNAME : STRING[10]
VAR_INPUT
	C : BYTE;
END_VAR
VAR
	pos: INT;
	i : INT;
END_VAR

(*
version 1.4		17. dec. 2008
programmer 		hugo
tested by		oscat

CHARNAME converts a Character code into its HTML character name
� is convterted to '�uml'
� is converted to 'euro'
the character itself is returned if no name is available for the character

*)
(* @END_DECLARATION := '0' *)
IF C <> 0 THEN
	(* construct search string from code followed by $ sign, also clear charname string*)
	CHARNAME := CHR_TO_STRING(C);
	CHARNAME := CONCAT(CHARNAME,'&');
	CHARNAME := CONCAT(';', CHARNAME);
	WHILE pos = 0 AND (i < 4) DO
		i := i + 1;
		pos := FIND(setup.CHARNAMES[i], CHARNAME);
	END_WHILE;
	IF pos > 0 THEN
		CHARNAME := MID(setup.CHARNAMES[i], 10, pos + 3);
		(* search for end of name and truncate *)
		pos := FIND(CHARNAME, ';');
		CHARNAME := LEFT(CHARNAME,pos - 1);
	ELSE
		CHARNAME := CHR_TO_STRING(C);
	END_IF;
ELSE
	CHARNAME := '';
END_IF;

(* revision history
hm	13. may. 2008	rev 1.0
	original version

hm	16. jun. 2008	rev 1.1
	changed nested call of concat for better compatibility

hm	19. oct. 2008	rev 1.2
	changes setup constants

hm	24. oct. 2008	rev 1.3
	new code for high performance

hm	17. dec. 2008	rev 1.4
	changed function chr to chr_to_string
*)

END_FUNCTION

(* @NESTEDCOMMENTS := 'Yes' *)
(* @PATH := '\/String' *)
(* @OBJECTFLAGS := '0, 8' *)
(* @SYMFILEFLAGS := '2048' *)
FUNCTION CHR_TO_STRING : STRING[1]
VAR_INPUT
	C : BYTE;
END_VAR
VAR
	PT : REF_TO BYTE;
END_VAR

(*
version 1.3	17. dec. 2008
programmer 	hugo
tested by	oscat

CHR creates a character from a byte input and stuffs it in a one character length string.

*)
(* @END_DECLARATION := '0' *)
PT := REF(CHR_TO_STRING);
PT^ := C;
pt := pt + 1;
pt^ := 0;

(* revision history
hm	16 jan 2007		rev 1.0
	original version

hm	4. feb. 2008	rev 1.1
	return string would not be terminated properly

hm	29. mar. 2008	rev 1.2
	changed STRING to STRING[1]

hm	17. dec. 2008	rev 1.3
	changed name of function from chr to chr_to_string
*)
END_FUNCTION

(* @NESTEDCOMMENTS := 'Yes' *)
(* @PATH := '\/String' *)
(* @OBJECTFLAGS := '0, 8' *)
(* @SYMFILEFLAGS := '2048' *)
FUNCTION CLEAN : STRING[STRING_LENGTH]
VAR_INPUT
	IN : STRING[STRING_LENGTH];
	CX : STRING[80];
END_VAR
VAR
	pos: INT := 1;
	stop: INT;
END_VAR

(*
version 1.0	18. jun. 2008
programmer 	hugo
tested by	oscat

Clean deletes all characters from a string except the ones specified in CX.

*)

(* @END_DECLARATION := '0' *)
(* copy input string *)
CLEAN := IN;
stop := LEN(in);
WHILE pos <= stop DO
	IF FIND(cx, MID(CLEAN, 1, pos)) > 0 THEN
		(* charcter found skip to next one *)
		pos := pos + 1;
	ELSE
		(* wrong chracter needs to be deleted *)
		CLEAN := DELETE(CLEAN, 1, pos);
		stop := stop - 1;	(* the string is one character shorter now *)
	END_IF;
END_WHILE;

(* revision history

hm		18. jun. 2008	rev 1.0
	original version

*)
END_FUNCTION

(* @NESTEDCOMMENTS := 'Yes' *)
(* @PATH := '\/String' *)
(* @OBJECTFLAGS := '0, 8' *)
(* @SYMFILEFLAGS := '2048' *)
FUNCTION CODE : BYTE
VAR_INPUT
	STR : STRING[STRING_LENGTH];
	POS : INT;
END_VAR
VAR
	PT : REF_TO BYTE;
END_VAR

(*
version 1.1	29. mar. 2008
programmer 	hugo
tested by		tobias

code extracts the code of a character at position POS of a string STR.

*)
(* @END_DECLARATION := '0' *)
IF pos < 1 OR pos > LEN(str) THEN
	CODE := 0;
	RETURN;
ELSE
	PT := REF(STR) + INT_TO_DWORD(pos - 1);
	CODE := pt^;
END_IF;

(* revision history
hm	9. mar. 2008	rev 1.0
	original version

hm	29. mar. 2008	rev 1.1
	changed STRING to STRING[STRING_LENGTH]
*)
END_FUNCTION

(* @NESTEDCOMMENTS := 'Yes' *)
(* @PATH := '\/String' *)
(* @OBJECTFLAGS := '0, 8' *)
(* @SYMFILEFLAGS := '2048' *)
FUNCTION COUNT_CHAR : INT
VAR_INPUT
	str : STRING[STRING_LENGTH];
	chr : BYTE;
END_VAR
VAR
	l: INT;
	pt : REF_TO BYTE;
	pos: INT;
END_VAR

(*
version 1.1	29. mar. 2008
programmer 		kurt
tested by		hugo

COUNT_CHAR counts how often a character CHAR occurs within a string STR.

*)
(* @END_DECLARATION := '0' *)
PT := REF(str);
l := LEN(str);
COUNT_CHAR := 0;
FOR pos := 1 TO l DO
	IF pt^ = CHR THEN COUNT_CHAR := COUNT_CHAR + 1; END_IF;
    PT := PT + 1;
END_FOR;

(* revision history
hm	29. feb 2008	rev 1.0
	original version

hm	29. mar. 2008	rev 1.1
	changed STRING to STRING[STRING_LENGTH]
*)
END_FUNCTION

(* @NESTEDCOMMENTS := 'Yes' *)
(* @PATH := '\/String' *)
(* @OBJECTFLAGS := '0, 8' *)
(* @SYMFILEFLAGS := '2048' *)
FUNCTION COUNT_SUBSTRING : INT
VAR_INPUT
   SEARCH : STRING;
   STR : STRING;
END_VAR
VAR
   pos : INT;
   size : INT;
END_VAR

(*
version 1.0	20. jan. 2011
programmed	kurt
tested by		tobias

count_substring returns the number of occurences of a substring in a string

*)
(* @END_DECLARATION := '0' *)
COUNT_SUBSTRING := 0;
size := LEN(SEARCH);
REPEAT
   pos := FIND(STR,SEARCH);
   IF pos > 0 THEN
      STR := REPLACE(STR, '', size,pos);
      COUNT_SUBSTRING := COUNT_SUBSTRING + 1;
   END_IF;
UNTIL pos = 0
END_REPEAT;

(* revision history
ks	20. jan. 2011	rev 1.0
	original version

*)

END_FUNCTION

(* @NESTEDCOMMENTS := 'Yes' *)
(* @PATH := '\/String' *)
(* @OBJECTFLAGS := '0, 8' *)
(* @SYMFILEFLAGS := '2048' *)
FUNCTION DEC_TO_BYTE : BYTE
VAR_INPUT
	DEC : STRING[10];
END_VAR
VAR
	pt : REF_TO BYTE;
	i: INT;
	X: BYTE;
	stop: INT;
END_VAR

(*
version 1.1	30. sep 2008
programmer 	hugo
tested by		oscat

DEC_TO_byte converts a decimal string into a byte.

*)
(* @END_DECLARATION := '0' *)
pt := REF(dec);
stop := LEN(DEC);
FOR I := 1 TO stop DO
	(* read the first character and subtract 48 to get value in decimal 0 = 48 *)
	x := pt^;
	(* calculate the value of the digit *)
	IF X > 47 AND x < 58 THEN
		DEC_TO_BYTE := DEC_TO_BYTE * 10 + X - 48;
	END_IF;
	pt := pt + 1;
END_FOR;

(* revision histroy
hm	20. jun. 2008	rev 1.0
	original release

hm	30. sep.2008	rev 1.1
	changed length of input string from 20 to 10
	corrected an error where decoding of characters 8 and 9 would fail

*)

END_FUNCTION

(* @NESTEDCOMMENTS := 'Yes' *)
(* @PATH := '\/String' *)
(* @OBJECTFLAGS := '0, 8' *)
(* @SYMFILEFLAGS := '2048' *)
FUNCTION DEC_TO_DWORD : DWORD
VAR_INPUT
	DEC : STRING[20];
END_VAR
VAR
	pt : REF_TO BYTE;
	i: INT;
	X: BYTE;
	stop: INT;
END_VAR

(*
version 1.1	30. sep. 2008
programmer 	hugo
tested by		oscat

DEC_TO_DWORD converts a decimal string into a DWORD.

*)
(* @END_DECLARATION := '0' *)
pt := REF(dec);
stop := LEN(dec);
FOR I := 1 TO stop DO
	(* read the first character and subtract 48 to get value in decimal 0 = 48 *)
	x := pt^;
	(* calculate the value of the digit *)
	IF X > 47 AND x < 58 THEN
		DEC_TO_DWORD := DEC_TO_DWORD * 10 + X - 48;
	END_IF;
	pt := pt + 1;
END_FOR;

(* revision histroy
hm	20. jun. 2008	rev 1.0
	original release

hm	30. sep. 2008	rev 1.1
	corrected an error where decoding of characters 8 and 9 would fail
*)

END_FUNCTION

(* @NESTEDCOMMENTS := 'Yes' *)
(* @PATH := '\/String' *)
(* @OBJECTFLAGS := '0, 8' *)
(* @SYMFILEFLAGS := '2048' *)
FUNCTION DEC_TO_INT : INT
VAR_INPUT
	DEC : STRING[10];
END_VAR
VAR
	pt : REF_TO BYTE;
	i: INT;
	X: BYTE;
	sign: BOOL;
	stop: INT;
END_VAR

(*
version 1.1	30. sep. 2008
programmer 	hugo
tested by	oscat

DEC_TO_INT converts a decimal string into an Integer.

*)
(* @END_DECLARATION := '0' *)
pt := REF(dec);
stop := LEN(dec);
FOR I := 1 TO stop DO
	(* read the first character and subtract 48 to get value in decimal 0 = 48 *)
	x := pt^;
	(* calculate the value of the digit *)
	IF X > 47 AND x < 58 THEN
		DEC_TO_INT := DEC_TO_INT * 10 + X - 48;
	ELSIF X = 45 AND DEC_TO_INT = 0 THEN
		sign := TRUE;
	END_IF;
	pt := pt + 1;
END_FOR;
IF sign THEN DEC_TO_INT := -DEC_TO_INT; END_IF;

(* revision histroy
hm	20. jun. 2008	rev 1.0
	original release

hm	30. sep. 2008	rev 1.1
	changed length of input string from 20 to 10
	corrected an error where decoding of characters 8 and 9 would fail
*)

END_FUNCTION

(* @NESTEDCOMMENTS := 'Yes' *)
(* @PATH := '\/String' *)
(* @OBJECTFLAGS := '0, 8' *)
(* @SYMFILEFLAGS := '2048' *)
FUNCTION DEL_CHARS : STRING[STRING_LENGTH]
VAR_INPUT
	IN : STRING[STRING_LENGTH];
	CX : STRING[80];
END_VAR
VAR
	pos: INT := 1;
	stop: INT;
END_VAR

(*
version 1.0	18. jun. 2008
programmer 	hugo
tested by	oscat

del_chars deletes all characters from a string which are specified in CX.

*)

(* @END_DECLARATION := '0' *)
(* copy input string *)
DEL_CHARS := IN;
stop := LEN(in);
WHILE pos <= stop DO
	IF FIND(cx, MID(DEL_CHARS, 1, pos)) > 0 THEN
		(* wrong chracter needs to be deleted *)
		DEL_CHARS := DELETE(DEL_CHARS, 1, pos);
		stop := stop - 1;	(* the string is one character shorter now *)
	ELSE
		(* charcter not found skip to next one *)
		pos := pos + 1;
	END_IF;
END_WHILE;

(* revision history

hm		18. jun. 2008	rev 1.0
	original version

*)
END_FUNCTION

(* @NESTEDCOMMENTS := 'Yes' *)
(* @PATH := '\/String' *)
(* @OBJECTFLAGS := '0, 8' *)
(* @SYMFILEFLAGS := '2048' *)
FUNCTION DT_TO_STRF : STRING
VAR_INPUT
	DTI : DT;
	MS : INT;
	FMT : STRING;
	LANG : INT;
END_VAR
VAR CONSTANT
	FILL : STRING[1] := '0';
	BLANK : STRING[1] := ' ';
END_VAR
VAR
	ly : INT;
	dx: DATE;
	fs: STRING[10];
	td: TOD;
	tmp : INT;
	pos : INT;
	f : INT;
END_VAR

(*
version 1.1	19. oct. 2008
programmer 	hugo
tested by	oscat

DT_TO_STRINGF converts a DATETIME input to a formatted string

*)
(* @END_DECLARATION := '0' *)
IF LANG < 1 THEN ly := language.DEFAULT; ELSE ly := MIN(language.LMAX, LANG); END_IF;

(* decode date and time information *)
dx := DT_TO_DATE(DTI);
td := DT_TO_TOD(DTI);

(* parse the format string *)
DT_TO_STRF := FMT;
pos := FIND(DT_TO_STRF, '#');
WHILE pos > 0 DO
	(* retrieve format identifier *)
	f := CODE(DT_TO_STRF, pos + 1);
	(* generate the return string according to the format character *)
	fs := '';
	CASE f OF
		65 : (* letter A retunrs the year in 4 digits *)
			fs := INT_TO_STRING(YEAR_OF_DATE(dx));
		66 : (* letter B returns the year in exactly 2 digits *)
			fs := RIGHT(INT_TO_STRING(YEAR_OF_DATE(dx)),2);
		67 : (* letter C returns the month with 1 or 2 digits *)
			fs := INT_TO_STRING(MONTH_OF_DATE(dx));
		68 : (* letter D returns the month with exactly 2 digits *)
			fs := INT_TO_STRING(MONTH_OF_DATE(dx));
			IF LEN(fs) < 2 THEN fs := CONCAT('0', fs); END_IF;
		69 : (* letter E returns the month with 3 characters *)
			fs := MONTH_TO_STRING(MONTH_OF_DATE(dx), ly, 3);
		70 : (* letter F returns the month with all characters *)
			fs := MONTH_TO_STRING(MONTH_OF_DATE(dx), ly, 0);
		71 : (* letter G returns the day with up to 2 digits *)
			fs := INT_TO_STRING(DAY_OF_MONTH(dx));
		72 : (* letter H returns the day of the month with exactly 2 digits *)
			fs := INT_TO_STRING(DAY_OF_MONTH(dx));
			IF LEN(fs) < 2 THEN fs := CONCAT(FILL, fs); END_IF;
		73 : (* letter I returns the weekday as the number 1..7 1 = monday *)
			fs := INT_TO_STRING(DAY_OF_WEEK(dx));
		74 : (* letter J returns the weekday in 2 character writing *)
			fs := WEEKDAY_TO_STRING(DAY_OF_WEEK(dx), ly, 2);
		75 : (* letter K returns the weekday with all characters *)
			fs := WEEKDAY_TO_STRING(DAY_OF_WEEK(dx), ly, 0);
		76 : (* letter L returns AM or PM for the given DateTime *)
			IF td >= TOD#12:00:00 THEN fs := 'PM'; ELSE fs := 'AM'; END_IF;
		77 : (* letter M returns the hour in 1 or 2 digit form 0..24h *)
			fs := INT_TO_STRING(HOUR(td));
		78 : (* letter N returns the hour in exactly 2 digit form 0..24h *)
			fs := INT_TO_STRING(HOUR(td));
			IF LEN(fs) < 2 THEN fs := CONCAT(FILL, fs); END_IF;
		79 : (* letter O returns the hour in 1 or 2 digit form 0..12h *)
			tmp := HOUR(td) MOD 12;
			IF tmp = 0 THEN tmp := 12; END_IF;
			fs := INT_TO_STRING(tmp);
		80 : (* letter P returns the hour in exactly 2 digit form 0..12h *)
			tmp := HOUR(td) MOD 12;
			IF tmp = 0 THEN tmp := 12; END_IF;
			fs := INT_TO_STRING(tmp);
			IF LEN(fs) < 2 THEN fs := CONCAT(FILL, fs); END_IF;
		81 : (* letter Q returns the minute of the hour in 1 or two digit form *)
			fs := INT_TO_STRING(MINUTE(td));
		82 : (* letter R returns the minute of the hour in exactly two digit form *)
			fs := INT_TO_STRING(MINUTE(td));
			IF LEN(fs) < 2 THEN fs := CONCAT(FILL, fs); END_IF;
		83 : (* letter S returns the second of the minute in 1 or two digit form *)
			fs := INT_TO_STRING(REAL_TO_INT(SECOND(td)));
		84 : (* letter T returns the second of the minute in exactly two digit form *)
			fs := INT_TO_STRING(REAL_TO_INT(SECOND(td)));
			IF LEN(fs) < 2 THEN fs := CONCAT(FILL, fs); END_IF;
		85 : (* letter U returns the milliseconds in 1 to 3 digits *)
			fs := INT_TO_STRING(MS);
		86 : (* letter V returns the milliseconds in exactly 3 digit form *)
			fs := INT_TO_STRING(MS);
			fs := CONCAT('00',fs);
			fs := RIGHT(fs, 3);
		87 : (* letter W returns the day of the month with exactly 2 digits first digit is filled with blank if necessary *)
			fs := INT_TO_STRING(DAY_OF_MONTH(dx));
			IF LEN(fs) < 2 THEN fs := CONCAT(BLANK, fs); END_IF;
		88 : (* letter X returns the month with exactly 2 digits first digit is filled with blank if necessary *)
			fs := INT_TO_STRING(MONTH_OF_DATE(dx));
			IF LEN(fs) < 2 THEN fs := CONCAT(BLANK, fs); END_IF;
		END_CASE;
	DT_TO_STRF := REPLACE(DT_TO_STRF, fs, 2, pos);
	pos := FIND(DT_TO_STRF, '#');
END_WHILE;

(* revision history
hm	7. oct. 2008	rev 1.0
	original version

hm	19. oct. 2008	rev 1.1
	changed language setup constants
*)

END_FUNCTION

(* @NESTEDCOMMENTS := 'Yes' *)
(* @PATH := '\/String' *)
(* @OBJECTFLAGS := '0, 8' *)
(* @SYMFILEFLAGS := '2048' *)
FUNCTION DWORD_TO_STRB : STRING[32]
VAR_INPUT
	IN : DWORD;
END_VAR
VAR
	pt : REF_TO BYTE;
	i: INT;
END_VAR

(*
version 1.3	20. jun. 2008
programmer 	hugo
tested by	oscat

DWORD_TO_STRINGB converts a DWORD to a String of Bits represented by '0' and '1' s.
The lowest order bit will be on the right and the high order bit on the left.

*)
(* @END_DECLARATION := '0' *)
(* pointer f�r die ausgabe ermitteln *)
pt := REF(DWORD_TO_STRB);
(* die 8 ausgabecharacter ermitteln und schreiben *)
FOR i := 1 TO 32 DO
	pt^:= BOOL_TO_BYTE(in.31) + 48;
	in := SHL(in,1);
	pt := pt + 1;
END_FOR;

(* der ausgabestring muss nochg mit 0 abgeschlossen werden *)
pt^ := 0;

(* revision history
hm		9.6.2007	rev 1.0
	original version

hm		15.dec 2007	rev 1.1
	changed code for better performance

hm	29. mar. 2008	rev 1.2
	changed STRING to STRING[32]

hm	20. jun. 2008	rev 1.3
	performance improvement

*)

END_FUNCTION

(* @NESTEDCOMMENTS := 'Yes' *)
(* @PATH := '\/String' *)
(* @OBJECTFLAGS := '0, 8' *)
(* @SYMFILEFLAGS := '2048' *)
FUNCTION DWORD_TO_STRF : STRING[20]
VAR_INPUT
	IN : DWORD;
	N : INT;
END_VAR

(*
version 1.0	26 jan 2007
programmer 	hugo
tested by		tobias

dword_to_strF converts a DWORD, BYTE or Word to a fixed length String.
the string will be filled with leading zeroes to achieve the fixed length, or if too long, the lowest digits will be used.
the maximum allowed length is 20 mdigits.

for example:	dword_to_strf(123,4) = '0123'
				dword_to_strf(123,2) = '23'
*)

(* @END_DECLARATION := '0' *)
(* limit N to max 20 characters *)
(* convert dword to string first and cut to length N *)
DWORD_TO_STRF := FIX(DWORD_TO_STRING(in),LIMIT(0,N,20),48,1);

(* revision history
hm	26. jan.2007	rev 1.0
	original version

hm	29. mar. 2008	rev 1.1
	changed STRING to STRING[20]
	limit the output string to max 20 digits
*)

END_FUNCTION

(* @NESTEDCOMMENTS := 'Yes' *)
(* @PATH := '\/String' *)
(* @OBJECTFLAGS := '0, 8' *)
(* @SYMFILEFLAGS := '2048' *)
FUNCTION DWORD_TO_STRH : STRING[8]
VAR_INPUT
	IN : DWORD;
END_VAR
VAR
	i : INT;
	temp : BYTE;
	pt : REF_TO BYTE;
END_VAR

(*
version 1.3	29. mar. 2008
programmer 	hugo
tested by	tobias

DWORD_TO_STRINGH converts a DWORD to a String of Hexadecimal represented by '0' .. '9' and 'A' .. 'F'.
The lowest order Character will be on the right and the high order Character on the left.

*)

(* @END_DECLARATION := '0' *)
(* read output adress to pointer *)
pt := REF(DWORD_TO_STRH) + 8;
(* wirte the closing byte for the string *)
pt^:= 0;

(* write the 8 hex characters backwards *)
FOR i := 1 TO 8 DO;
	(* decrement the pointer *)
	pt := pt - 1;
	(* read the lowest order hex value *)
	temp := DWORD_TO_BYTE(in AND 16#0000000F);
	(* convert value to hex character *)
	IF temp <= 9 THEN temp := temp + 48; ELSE temp := temp + 55; END_IF;
	(* write character to output string *)
	PT^ := temp;
	(* shift in for nect hex character *)
	in := SHR(in,4);
END_FOR;

(* code beofre rev 1.2
FOR i := 1 TO 8 DO
	X := DWORD_TO_BYTE(in AND 2#1111);
	IF X <= 9 THEN X := X + 48; ELSE X := X + 55; END_IF;
	Cx := CHR(X);
	temp := CONCAT(Cx, temp);
	in := SHR(in,4);
END_FOR;
DWORD_TO_STRH := temp;
*)

(* revision history
hm	9. jun. 2007	rev 1.0
	original version

hm	11. sep. 2007	rev 1.1
	changed coding for compatibility with twincat, concat cannot support a function as an argument.

hm	15. dec. 2007	rev 1.2
	changed code for better performance

hm	29. mar. 2008	rev 1.3
	changed STRING to STRING[8]

*)

END_FUNCTION

(* @NESTEDCOMMENTS := 'Yes' *)
(* @PATH := '\/String' *)
(* @OBJECTFLAGS := '0, 8' *)
(* @SYMFILEFLAGS := '2048' *)
FUNCTION EXEC : STRING[STRING_LENGTH]
VAR_INPUT
	str : STRING[STRING_LENGTH];
END_VAR
VAR
	pos: INT;
	R1: REAL;
	R2: REAL;
	operator: STRING[10];
END_VAR

(*
version 1.4	29. mar. 2008
programmer 	hugo
tested by		tobias

exec executes a mathematical term and returns the result as a string
the term can only be a simple term without brackets and only one operator
allowed operastors are: (+, -, *, /, ^, sqrt, sin, cos, tan).

*)
(* @END_DECLARATION := '0' *)
(* extract both numbers and operator *)
EXEC := UPPERCASE(TRIM(str));

pos := FINDB_NONUM(EXEC);
IF pos > 1 THEN R1 := STRING_TO_REAL(LEFT(EXEC,pos-1)); END_IF;
R2 := STRING_TO_REAL(RIGHT(EXEC,LEN(EXEC)-pos));
EXEC := LEFT(EXEC,pos);
pos := FINDB_NUM(EXEC);
operator := RIGHT(EXEC,LEN(EXEC) - pos);
IF operator = '' AND LEN(str) = 0 THEN
	EXEC := '';
	RETURN;
ELSIF operator = '' THEN
	EXEC := str;
	RETURN;
END_IF;
IF operator = '^' THEN
	EXEC := REAL_TO_STRING(EXPT(R1, R2));
ELSIF operator = 'SQRT' THEN
	EXEC := REAL_TO_STRING(SQRT(R2));
ELSIF operator = 'SIN' THEN
	EXEC := REAL_TO_STRING(SIN(r2));
ELSIF operator = 'COS' THEN
	EXEC := REAL_TO_STRING(COS(r2));
ELSIF operator = 'TAN' THEN
	EXEC := REAL_TO_STRING(TAN(R2));
ELSIF operator = '*' THEN
	EXEC := REAL_TO_STRING(R1 * R2);
ELSIF operator = '/' THEN
	IF R2 <> 0 THEN EXEC := REAL_TO_STRING(R1 / R2); ELSE EXEC := 'ERROR'; END_IF;
ELSIF operator = '+' THEN
	EXEC := REAL_TO_STRING(r1 + r2);
ELSIF operator = '-' THEN
	EXEC := REAL_TO_STRING(r1 - r2);
ELSE
	EXEC := 'ERROR';
END_IF;

IF EXEC = 'ERROR' THEN
	RETURN;
(* some systems deliver integer instead of real *)
ELSIF FIND(EXEC,'.') = 0 THEN
	EXEC := CONCAT(EXEC, '.0');
(* some systems deliver n. instead of n.0 ! *)
ELSIF RIGHT(EXEC,1) = '.' THEN
	EXEC := CONCAT(EXEC,'0');
END_IF;

(* revision history

hm 	6.feb 2007		rev 1.1
	cos has to be written in uppercase
	divide by 0 will return an error

hm	5. mar. 2008	rev 1.2
	add a 0 to the string if a '.' is at the end of the string

hm	20. mar. 2008	rev 1.3
	make sure the function always returns a real value in the form of x.y

hm	29. mar. 2008	rev 1.4
	changed STRING to STRING[STRING_LENGTH]
*)
END_FUNCTION

(* @NESTEDCOMMENTS := 'Yes' *)
(* @PATH := '\/String' *)
(* @OBJECTFLAGS := '0, 8' *)
(* @SYMFILEFLAGS := '2048' *)
FUNCTION FILL : STRING[STRING_LENGTH]
VAR_INPUT
	C : BYTE;
	L : INT;
END_VAR
VAR
	i: INT;
	sx: STRING[1];
END_VAR

(*
version 1.1	17. dec. 2008
programmer 	hugo
tested by		tobias

the function fill creates a string at length L of characters C.

*)
(* @END_DECLARATION := '0' *)
Sx := CHR_TO_STRING(c);
(* limit L to maximum 80 characters the length of a standard string *)
L := LIMIT(0,L,STRING_LENGTH);
(* create a string of characters to be connected to str *)
FOR i := 1 TO 8 DO
	FILL := CONCAT(FILL,FILL);
	IF L.7 THEN FILL := CONCAT(FILL,Sx); END_IF;
	L := SHL(L,1);
END_FOR;

(* revision histroy
hm	29. mar. 2008	rev 1.0
	original release

hm	17. dec. 2008	rev 1.1
	changed function chr to chr_to_string

*)
END_FUNCTION

(* @NESTEDCOMMENTS := 'Yes' *)
(* @PATH := '\/String' *)
(* @OBJECTFLAGS := '0, 8' *)
(* @SYMFILEFLAGS := '2048' *)
FUNCTION FIND_CHAR : INT
VAR_INPUT
	str : STRING[STRING_LENGTH];
	pos : INT;
END_VAR
VAR
	i: INT;
	pt : REF_TO ARRAY[1..255] OF BYTE;
	stop: INT;
	X: BYTE;
END_VAR

(*
version 1.3	21. oct. 2008
programmer 	hugo
tested by	tobias

find_char searches str and returns the starting position of the first character that is not a control character.
control characters are the ascii character 00 .. 31 and 127

*)
(* @END_DECLARATION := '0' *)
pt := REF(str);
stop := LEN(str);
FOR i := MAX(pos,1) TO stop DO;
	X := pt^[i];
	IF X > 31 AND ((setup.EXTENDED_ASCII AND X <> 127) OR (NOT setup.EXTENDED_ASCII AND X < 127)) THEN
		FIND_CHAR := i;
		RETURN;
	END_IF;
END_FOR;
FIND_CHAR := 0;

(* revision history
hm	29. feb 2008	rev 1.0
	original version

hm	26. mar. 2008	rev 1.1
	char will now accept extended ascii

hm	29. mar. 2008	rev 1.2
	changed STRING to STRING[STRING_LENGTH]

hm	21. oct. 2008	rev 1.3
	changes setup constants
	optimized code
*)

END_FUNCTION

(* @NESTEDCOMMENTS := 'Yes' *)
(* @PATH := '\/String' *)
(* @OBJECTFLAGS := '0, 8' *)
(* @SYMFILEFLAGS := '2048' *)
FUNCTION FIND_CTRL : INT
VAR_INPUT
	str : STRING[STRING_LENGTH];
	pos : INT;
END_VAR
VAR
	i: INT;
	pt : REF_TO ARRAY[1..255] OF BYTE;
	stop: INT;
	x: BYTE;
END_VAR
